# B&R Automation Studio project PloterCNC (part 5)

```c
	return fmi2OK;
}
/* END: fmi2SetString */
/*****************************************************************************/

/*****************************************************************************/
/* BEGIN: fmi2GetFMUstate */
/*****************************************************************************/
/* Storage structure:
		State id (hard coded value)
		Data length (bytes)
		ModelInstance
		Real data storage
		Integer data storage
		Real backup data storage (only for ME)
		Jacobian storage
		Error code
		String storage
*/
#define FMUStateID 983472598

fmi2Status fmi2GetFMUstate (
	fmi2Component	c,
	fmi2FMUstate*	FMUstate
)
{
	ModelInstance* comp = (ModelInstance *)c;
	char *cur;
	fmi2Real *rcur;
	M_INT i,j,*icur,wsto,ssto,jsto,totsto;

	if (invalidState(comp, "fmi2GetFMUstate", modelInitialized))
		return fmi2Error;

	if(comp->fmuType==fmi2ModelExchange)
		wsto = NUMBER_OF_REALS*sizeof(fmi2Real);
	else
		wsto = 0;

#ifdef FMI2_PROVIDES_DERIVATIVES
	jsto=( (1+NDIFF+NINP)*(NDIFF+NOUT) + NIUNK*(NIKNO+1) )*sizeof(fmi2Real);
#else
	jsto=0;
#endif

	ssto=0;
	for(i=0;i<NUMBER_OF_STRINGS;i++)
		if(comp->s[i])
			ssto+=strlen(comp->s[i])+1;
		else
			ssto++;

	totsto = 2*sizeof(M_INT) +
				sizeof(ModelInstance) +
				NUMBER_OF_REALS*sizeof(fmi2Real) +
				NUMBER_OF_INTEGERS*sizeof(M_INT) +
				wsto +
				jsto +
				sizeof(M_INT) +
				ssto;

	/* Verify that previously allocated FMU state is of sufficient size */
	if(*FMUstate) {
		icur=(M_INT *)(*FMUstate);
		if(icur[0]!=FMUStateID) {
			/* FMUstate pointer is not previously allocated in this routine
				so no way to verify the size */
			compLog(compEnv, comp->instanceName, fmi2Warning, "warning",
				"fmi2GetFMUstate: called with non-NULL state pointer of unknown size. Assuming sufficiently large.");
		}
		else if(icur[1]<totsto) {
			comp->functions.freeMemory(*FMUstate);
			*FMUstate=NULL;
		}
	}

	if(*FMUstate==NULL)
		FMUstate[0] = (fmi2FMUstate)comp->functions.allocateMemory(1,totsto);

	cur = (char *)(*FMUstate);

	icur = (M_INT *)cur;
	icur[0] = FMUStateID;
	icur[1] = totsto;
	cur += 2*sizeof(M_INT);

	memcpy(cur,comp,sizeof(ModelInstance));
	cur += sizeof(ModelInstance);

	rcur = (fmi2Real*)cur;
	for (i=0;i<NUMBER_OF_REALS;i++)	rcur[i] = comp->S.w[i];
	cur += NUMBER_OF_REALS*sizeof(fmi2Real);

	icur = (M_INT *)cur;
	for (i=0;i<NUMBER_OF_INTEGERS;i++) icur[i] = comp->S.iw[i];
	cur += NUMBER_OF_INTEGERS*sizeof(M_INT);

	if(comp->fmuType==fmi2ModelExchange) {
		rcur = (fmi2Real*)cur;
		for (i=0;i<NUMBER_OF_REALS;i++)	rcur[i] = comp->S.wset[i];
		cur += NUMBER_OF_REALS*sizeof(fmi2Real);
	}

#ifdef FMI2_PROVIDES_DERIVATIVES
	rcur = (fmi2Real*)cur;
	for (i=0;i<(1+NDIFF+NINP)*(NDIFF+NOUT);i++)	rcur[i] = comp->Jacobian[i];
	cur += (1+NDIFF+NINP)*(NDIFF+NOUT)*sizeof(fmi2Real);

	rcur = (fmi2Real*)cur;
	for (i=0;i<NIUNK*NIKNO;i++)	rcur[i] = comp->initJacobian[i];
	cur += NIUNK*NIKNO*sizeof(fmi2Real);

	rcur = (fmi2Real*)cur;
	for (i=0;i<NIUNK;i++)	rcur[i] = comp->initRes[i];
	cur += NIUNK*sizeof(fmi2Real);
#endif

	icur = (M_INT *)cur;
	icur[0] = errorOccured;
	cur += sizeof(M_INT);

	for(i=0;i<NUMBER_OF_STRINGS;i++) {
		if(comp->s[i]) {
			for(j=0;comp->s[i][j]!='\0';j++)
				*(cur++)=comp->s[i][j];
		}
		*(cur++)='\0';
	}

	return fmi2OK;
}
/* END: fmi2GetFMUstate */
/*****************************************************************************/

/*****************************************************************************/
/* BEGIN: fmi2SetFMUstate */
/*****************************************************************************/
fmi2Status fmi2SetFMUstate (fmi2Component	c,
							fmi2FMUstate	FMUstate) {
	ModelInstance* comp = (ModelInstance *)c;
	char *cur;
	fmi2String *scur;
	fmi2Real *rcur,*wcur,*jcur1,*jcur2,*jcur3;
	M_INT i,j,l,*icur;

	if (invalidState(comp, "fmi2SetFMUstate", modelInitialized))
		return fmi2Error;

	cur = (char *)FMUstate;
	icur = (M_INT *)cur;
	if(icur[0]!=FMUStateID) {
		compLog(compEnv, comp->instanceName, fmi2Error, "error",
			"fmi2SetFMUstate: called with invalid FMUstate");
		return(fmi2Error);
	}
	cur += 2*sizeof(M_INT);

	rcur = comp->S.w;
	icur = comp->S.iw;
	wcur = comp->S.wset;
	jcur1 = comp->Jacobian;
	jcur2 = comp->initJacobian;
	jcur3 = comp->initRes;
	scur = comp->s;
	memcpy(comp,cur,sizeof(ModelInstance));
	comp->S.w  = rcur;
	comp->S.iw = icur;
	comp->S.wset = wcur;
	comp->Jacobian = jcur1;
	comp->initJacobian = jcur2;
	comp->initRes = jcur3;
	comp->s = scur;
	cur += sizeof(ModelInstance);

	rcur = (fmi2Real *)cur;
	for(i=0;i<NUMBER_OF_REALS;i++) comp->S.w[i] = rcur[i];
	cur += NUMBER_OF_REALS*sizeof(fmi2Real);

	icur = (M_INT *)cur;
	for (i=0;i<NUMBER_OF_INTEGERS;i++) comp->S.iw[i] = icur[i];
	cur += NUMBER_OF_INTEGERS*sizeof(M_INT);

	if(comp->fmuType==fmi2ModelExchange) {
		rcur = (fmi2Real *)cur;
		for(i=0;i<NUMBER_OF_REALS;i++) comp->S.wset[i] = rcur[i];
		cur += NUMBER_OF_REALS*sizeof(fmi2Real);
	}
	else
		comp->S.wset = NULL;

#ifdef FMI2_PROVIDES_DERIVATIVES
	rcur = (fmi2Real*)cur;
	for (i=0;i<(1+NDIFF+NINP)*(NDIFF+NOUT);i++)	comp->Jacobian[i] = rcur[i];
	cur += (1+NDIFF+NINP)*(NDIFF+NOUT)*sizeof(fmi2Real);

	rcur = (fmi2Real*)cur;
	for (i=0;i<NIUNK*NIKNO;i++)	comp->initJacobian[i] = rcur[i];
	cur += NIUNK*NIKNO*sizeof(fmi2Real);

	rcur = (fmi2Real*)cur;
	for (i=0;i<NIUNK;i++)	comp->initRes[i] = rcur[i];
	cur += NIUNK*sizeof(fmi2Real);
#else
	comp->Jacobian = NULL;
	comp->initJacobian = NULL;
	comp->initRes = NULL;
#endif

	icur = (M_INT *)cur;
	errorOccured = icur[0];
	cur += sizeof(M_INT);

	for(i=0;i<NUMBER_OF_STRINGS;i++) {
		l=(comp->s[i]) ? strlen(comp->s[i]) : 0;
		j=strlen(cur);
		if(j>l) {
			if(comp->s[i]) comp->functions.freeMemory((char *)comp->s[i]);
			comp->s[i]=(fmi2String)comp->functions.allocateMemory(1,j+1);
		}
		strcpy((char *)comp->s[i],cur);
		cur += j+1;
	}

	return fmi2OK;
}
/* END: fmi2SetFMUstate */
/*****************************************************************************/

/*****************************************************************************/
/* BEGIN: fmi2FreeFMUstate */
/*****************************************************************************/
fmi2Status fmi2FreeFMUstate(fmi2Component c,
							fmi2FMUstate* FMUstate) {
	ModelInstance* comp = (ModelInstance *)c;
	M_INT *icur;

	if (invalidState(comp, "fmi2FreeFMUstate",
		modelInstantiated|modelInitialized|modelTerminated|modelError))
		return fmi2Error;

	if( *FMUstate ) {
		icur = (M_INT *)(*FMUstate);
		if(icur[0]!=FMUStateID)
			compLog(compEnv, comp->instanceName, fmi2Warning, "warning",
				"fmi2FreeFMUstate: called with invalid FMUstate");
		comp->functions.freeMemory(*FMUstate);
	}

	*FMUstate = NULL;

	return fmi2OK;
}
/* END: fmi2FreeFMUstate */
/*****************************************************************************/

/*****************************************************************************/
/* BEGIN: fmi2SerializedFMUstateSize */
/*****************************************************************************/
fmi2Status fmi2SerializedFMUstateSize(	fmi2Component	c,
										fmi2FMUstate	FMUstate,
										size_t			*size) {
	ModelInstance* comp = (ModelInstance *)c;
	M_INT *icur;

	if (invalidState(comp, "fmi2SerializedFMUstateSize", modelInitialized))
		return fmi2Error;

	icur = (M_INT *)FMUstate;
	if(icur[0]!=FMUStateID) {
		compLog(compEnv, comp->instanceName, fmi2Error, "error",
			"fmi2SerializedFMUstateSize: called with invalid FMUstate");
		return(fmi2Error);
	}
	*size = (size_t)icur[1];

	return fmi2OK;
}
/* END: fmi2SerializedFMUstateSize */
/*****************************************************************************/

/*****************************************************************************/
/* BEGIN: fmi2SerializeFMUstate */
/*****************************************************************************/
fmi2Status fmi2SerializeFMUstate(fmi2Component		c,
								fmi2FMUstate		FMUstate,
								fmi2Byte 			serializedState[],
								size_t				size) {
	ModelInstance* comp = (ModelInstance *)c;
	M_INT *icur;

	if (invalidState(comp, "fmi2SerializeFMUstate", modelInitialized))
		return fmi2Error;

	icur = (M_INT *)FMUstate;
	if(icur[0]!=FMUStateID) {
		compLog(compEnv, comp->instanceName, fmi2Error, "error",
			"fmi2SerializedFMUstate: called with invalid FMUstate");
		return fmi2Error;
	}
	if(icur[1]>(M_INT)size) {
		compLog(compEnv, comp->instanceName, fmi2Error, "error",
			"fmi2SerializedFMUstate: called with size not sufficient to contain FMUstate");
		return fmi2Error;
	}
	memcpy(serializedState, FMUstate, size);

	return fmi2OK;
}
/* END: fmi2SerializeFMUstate */
/*****************************************************************************/

/*****************************************************************************/
/* BEGIN: fmi2DeSerializeFMUstate */
/*****************************************************************************/
fmi2Status fmi2DeSerializeFMUstate(	fmi2Component	c,
									const fmi2Byte	serializedState[],
									size_t			size,
									fmi2FMUstate	*FMUstate) {
	ModelInstance* comp = (ModelInstance *)c;
	M_INT *icur;

	if (invalidState(comp, "fmi2DeSerializeFMUstate", modelInitialized))
		return fmi2Error;

	icur = (M_INT *)serializedState;
	if(icur[0]!=FMUStateID) {
		compLog(compEnv, comp->instanceName, fmi2Error, "error",
			"fmi2DeSerializedFMUstate: called with serializedState not containing valid FMUstate");
		return fmi2Error;
	}
	if(icur[1]>(M_INT)size) {
		compLog(compEnv, comp->instanceName, fmi2Error, "error",
			"fmi2SerializedFMUstate: called with size not sufficient to contain serializedState");
		return fmi2Error;
	}
	FMUstate[0] = (fmi2FMUstate)comp->functions.allocateMemory(1,size);
	memcpy(*FMUstate, serializedState, size);

	return fmi2OK;
}
/* END: fmi2DeSerializeFMUstate */
/*****************************************************************************/

/*****************************************************************************/
/* BEGIN: fmi2GetDirectionalDerivative */
/*****************************************************************************/
fmi2Status fmi2GetDirectionalDerivative(	fmi2Component			c,
										const fmi2ValueReference	vUnknown_ref[],
										size_t						nUnknown,
										const fmi2ValueReference	vKnown_ref[],
										size_t						nKnown,
										const fmi2Real				dvKnown[],
										fmi2Real					dvUnknown[]) {
#ifdef FMI2_PROVIDES_DERIVATIVES
	int i, j, k, row, col, offset;
	fmi2Status sts;
	fmi2ValueReference vrs, vrd;
	ModelInstance* comp = (ModelInstance *)c;

	if (invalidState(comp, "fmi2GetDirectionalDerivatives", modelInstantiated|modelInitialized))
		return fmi2Error;
	if (nKnown>0 && nullPointer(comp, "fmi2GetDirectionalDerivative", "vKnown_ref[]", vKnown_ref))
		return fmi2Error;
	if (nUnknown>0 && nullPointer(comp, "fmi2GetDirectionalDerivative", "vUnknown_ref[]", vUnknown_ref))
		return fmi2Error;
	if (nKnown>0 && nullPointer(comp, "fmi2GetDirectionalDerivative", "dvKnown[]", dvKnown))
		return fmi2Error;

	sts = syncModel(comp,"fmi2GetDirectionalDerivative");
	if ( sts!=fmi2OK ) return sts;

	/* Initialize unknown vector */
	for (i=0; i<nUnknown; i++) dvUnknown[i] = 0.;

	/* Get Jacobian information, dimensions, data, etc? */
	if(!comp->jsynced) {
		if(comp->initializeMode)
			initjac(comp->S.w[0],&(comp->S.w[1]),&(comp->S.w[NEQ+NPAR+1]),comp->initRes,comp->initJacobian);
		else
			intjac(comp->S.w[0],&(comp->S.w[1]),&(comp->S.w[NEQ+NPAR+1]),comp->Jacobian);
		comp->jsynced = fmi2True;
	}

	/* Order of value references :
	t, #states, #index-1(inps), #discrete, #params, #derivs, #events */

	/* Start the computation loop */
	if (comp->initializeMode) {
		offset = NIKNO;
		for (i=0; i<nKnown; i++) {
			/* Check the seed */
			if (dvKnown[i]!=0) {
				vrs = vKnown_ref[i];
				/* assert(vr>=0 && vr<NUMBER_OF_REALS); */
				col = -1;
				for (k=0; k<NIKNO; k++)
					if (vrs==vrIknowns[k]) {
						col = k;
						break;
					}
				/* Compute column i */
				for (j=0; j<nUnknown; j++) {
					vrd = vUnknown_ref[j];
					/* assert(vrd>=0 && vrd<NUMBER_OF_REALS); */
					if ( vrd==vrs ) {
						dvUnknown[j] += 1.0;
					}
					else if(col!=-1) {
						for (k=0; k<NIUNK; k++)
							if (vrd==vrIunknowns[k]) {
								dvUnknown[j] += dvKnown[i]*comp->initJacobian[k*offset+col];
								break;
							}
					}
				}
			}
		}
	}
	else {
		offset = 1+NDIFF+NINP;
		for (i=0; i<nKnown; i++) {
			/* Check the seed */
			if (dvKnown[i]!=0) {
				vrs = vKnown_ref[i];
				/* assert(vr>=0 && vr<NUMBER_OF_REALS); */
				/* Check that vKnown_ref[i] is a state or input */
				if ( vrs==0 || (vrs>=vrStates[0] && vrs<vrStates[0]+NDIFF) )
					col = vrs;
				else if(vrs>=1+NDIFF+NIX1-NINP && vrs<1+NDIFF+NIX1)
					col = vrs-(NIX1-NINP);
				else
					return fmi2Error;
				/* Compute column i */
				for (j=0; j<nUnknown; j++) {
					vrd = vUnknown_ref[j];
					/* assert(vrd>=0 && vrd<NUMBER_OF_REALS); */
					/* Check if vrd is a derivative or an output,
					it could also be an output that's a state */
					if ( vrd>=vrDers[0] && vrd<vrDers[0]+NDIFF ) {
						row = vrd-vrDers[0];
						dvUnknown[j] += dvKnown[i]*comp->Jacobian[row*offset+col];
					}
					else if( vrd>=vrStates[0] && vrd<vrStates[0]+NDIFF ) {
						if ( vrd==vrs ) dvUnknown[j] += 1.0;
					}
					else {
						for (k=0; k<NOUT; k++)
							if (vrd==vrOuts[k]) {
								/* refval-t-states+derivs: vrd-1-NDIFF+NDIFF */
								row = vrd-1;
								dvUnknown[j] += dvKnown[i]*comp->Jacobian[row*offset+col];
								break;
							}
						if (k==NOUT) return fmi2Error;
					}
				}
			}
		}
	}
	return fmi2OK;
#else
	/* Compiler warning fix */
	int i=nUnknown+nKnown;
	void *tmp;
	tmp=(void *)vUnknown_ref;
	tmp=(void *)vKnown_ref;
	tmp=(void *)dvKnown;
	tmp=(void *)dvUnknown;
	if(i>0) tmp=(void *)c;
	i=((int *)tmp)[0];
	/* End compiler warning fix */
	return fmi2Error;
#endif
}
/* END: fmi2GetDirectionalDerivative */
/*****************************************************************************/

#if NCON>0 && defined(WMI_PROJECTION)
/*****************************************************************************/
/* BEGIN: fmi2Projection */
/*****************************************************************************/
fmi2Status fmi2Projection(	fmi2Component	c,
								fmi2Real	P[],
								fmi2Real	projectionTolerance,
								size_t	iterationLimit,
								fmi2Boolean	apply) {
	int i;
	fmi2Status sts;
	fmi2Real S2[NDIFF];

	ModelInstance* comp = (ModelInstance *)c;

	if (invalidState(comp, "fmi2Projection", modelInstantiated|modelInitialized))
		return fmi2Error;

	sts = syncModel(comp,"fmi2Projection");
	if ( sts!=fmi2OK ) return sts;

	for(i=0;i<NDIFF;i++) S2[i] = comp->S.w[i+1];
	i=Projection(comp->S.w[0], &comp->S.w[1], projectionTolerance,
		iterationLimit, NULL, comp->S.psto);
	if( i!=0 ){
		/* Restore state */
		for(i=0;i<NDIFF;i++) comp->S.w[i+1]=S2[i];
		return fmi2Discard;
	}
	for(i=0;i<NDIFF;i++) P[i] = comp->S.w[i+1]-S2[i];

	if( !apply ){
		for(i=0;i<NDIFF;i++) comp->S.w[i+1]=S2[i];
	}

	return fmi2OK;
}
/* END: fmi2Projection */
/*****************************************************************************/

/*****************************************************************************/
/* BEGIN: fmi2ProjectionStep: No longer supported */
/*****************************************************************************/
fmi2Status fmi2ProjectionStep(  fmi2Component	c,
								fmi2Real	S[]) {
	UNUSED(c);
	UNUSED(S);
	return fmi2Error;
}
/* END: fmi2ProjectionStep */
/*****************************************************************************/

/*****************************************************************************/
/* BEGIN: fmi2Constraint */
/*****************************************************************************/
fmi2Status fmi2Constraint(	fmi2Component	c,
								fmi2Real	C[]) {
	int cb, cr, nblk;
	fmi2Real blkdata[2];
	fmi2Status sts;

	ModelInstance* comp = (ModelInstance *)c;

	if (invalidState(comp, "fmi2Constraint", modelInstantiated|modelInitialized))
		return fmi2Error;

	sts = syncModel(comp,"fmi2Constraint");
	if ( sts!=fmi2OK ) return sts;

	/* Iterate over Residual blocks */
	Rblkp(comp->S.w[0], &comp->S.w[1], blkdata, 0, 0);
	nblk = (int)(blkdata[0]);
	cr = 0;
	for(cb=1;cb<=nblk;cb++) {
		Rblkp(comp->S.w[0], &comp->S.w[1], &C[cr], cb, 3);
		Rblkp(comp->S.w[0], &comp->S.w[1], blkdata, cb, 1);
		cr += (int)(blkdata[0]);
	}

	return fmi2OK;
}
/* END: fmi2Constraint */
/*****************************************************************************/

/*****************************************************************************/
/* BEGIN: fmi2ConstraintJacobian: No longer supported */
/*****************************************************************************/
fmi2Status fmi2ConstraintJacobian(	fmi2Component	c,
										fmi2Real	J[]) {

	/* If this function is required at some point, the code will need to be
	modified to fill in the ncon x ndiff Matrix using a sequence of calls to
	the block-based Jacobian. It is known that this will provide 0 entries
	for block dependencies on vars from a prior block, but this will only
	slow convergence of a newton approach, and be irrelevant when sufficiently
	close to the solution manifold */
	UNUSED(c);
	UNUSED(J);
	return fmi2Error;
}
/* END: fmi2ConstraintJacobian */
/*****************************************************************************/
#endif

#ifdef FMI2_COSIMULATION
/*****************************************************************************
 * FMI functions: only for FMI Co-Simulation 2.0
 *****************************************************************************/
/*****************************************************************************/
/* BEGIN: fmi2SetRealInputDerivatives */
fmi2Status fmi2SetRealInputDerivatives(	fmi2Component			c,
										const fmi2ValueReference vr[],
										size_t					nvr,
										const fmi2Integer		order[],
										const fmi2Real			value[]) {
	ModelInstance* comp = (ModelInstance *)c;

	if (invalidState(comp, "fmi2SetRealInputDerivatives", modelInitialized))
		return fmi2Error;
	if (comp->loggingOn)
		compLog(compEnv, comp->instanceName, fmi2OK, "log",
				"fmi2SetRealInputDerivatives: nvr= %d", nvr);

	UNUSED(vr);
	UNUSED(order);
	UNUSED(value);
	compLog(NULL, comp->instanceName, fmi2Error, "warning",
			"fmi2SetRealInputDerivatives: ignoring function call."
			" This model cannot interpolate inputs: canInterpolateInputs = \"fmi2False\"");

	return fmi2Warning;
}
/* END: fmi2SetRealInputDerivatives */
/*****************************************************************************/

/*****************************************************************************/
/* BEGIN: fmi2GetRealOutputDerivatives */
fmi2Status fmi2GetRealOutputDerivatives(fmi2Component			c,
										const fmi2ValueReference vr[],
										size_t					nvr,
										const fmi2Integer		order[],
										fmi2Real				value[]) {
	int i;
	ModelInstance* comp = (ModelInstance *)c;

	if (invalidState(comp, "fmi2GetRealOutputDerivatives", modelInitialized))
		return fmi2Error;
	if (comp->loggingOn)
		compLog(compEnv, comp->instanceName, fmi2OK, "log",
				"fmi2GetRealOutputDerivatives: nvr= %d",	nvr);

	UNUSED(vr);
	UNUSED(order);
	compLog(NULL, comp->instanceName, fmi2Error, "warning",
			"fmi2GetRealOutputDerivatives: ignoring function call."
			" This model cannot compute derivatives of outputs: MaxOutputDerivativeOrder=\"0\"");

	for (i=0; i<(int)nvr; i++) value[i] = 0;

	return fmi2Warning;
}
/* END: fmi2GetRealOutputDerivatives */
/*****************************************************************************/

#define MAX_STEP  1.00000000000000000e-04

/*****************************************************************************/
/* BEGIN: fmi2DoStep */
fmi2Status fmi2DoStep(  fmi2Component	c,
						fmi2Real		currentCommunicationPoint,
						fmi2Real		communicationStepSize,
						fmi2Boolean		newStep) {

	ModelInstance* comp	= (ModelInstance *)c;
	int		i;
	double	h;
#if NEVT>0
	M_INT *modes;
	double	prevEventIndicators[max(NEVT, 1)];
#endif

	if (invalidState(comp, "fmi2DoStep", modelInitialized)) return fmi2Error;

	if (comp->loggingOn)
		compLog(compEnv, comp->instanceName, fmi2OK, "log", "fmi2DoStep: "
				"currentCommunicationPoint = %g, "
				"communicationStepSize = %g, "
				"newStep = fmi2%s",
				currentCommunicationPoint, communicationStepSize, newStep ? "True" : "False");

	if (comp->stopTimeDefined && currentCommunicationPoint+communicationStepSize > comp->stopTime) {
		comp->state = modelError;
		return fmi2Error;
	}

#if NPAR>0
	if(pchange) {
		SolverInitialize(&(comp->S));
		pchange=0;
		if (errorOccured>0) {
			setVidError(comp,NULL);
			if (comp->fptr) {
				writeErrorToFile(comp->fptr,NULL);
				comp->fptr = NULL;
			}
			comp->state = modelTerminated;
			logMessage(comp, "fmi2DoStep", "error", fmi2Error);
			return fmi2Error;
		}
		else if(errorOccured<0) {
			logMessage(comp, "fmi2DoStep", "warning", fmi2Warning);
			errorOccured=0;
		}
	}
#endif

#if NEVT>0
	/* Run to get initial event indicators */
	eev(comp->S.w[0],&(comp->S.w[1]),&(comp->S.w[1]),prevEventIndicators);
	modes=comp->S.iw;
	ComputeEventIndicators(prevEventIndicators,&(comp->S.w[1]),modes,
		&modes[3*NEVT],&modes[2*NEVT],&modes[4*NEVT]);
#endif

	comp->S.w[0] = currentCommunicationPoint;
	if( currentCommunicationPoint < (comp->lastSuccessfulTime-10.*ULP1) )
		comp->lastStepSize = -1.;
	h = ( comp->lastStepSize<0. ) ? communicationStepSize/100. : comp->lastStepSize;
	warningOccured=0;
	/* Call the variable step integrator */
	i = Integrate(comp->S.w,comp->S.iw,currentCommunicationPoint+communicationStepSize,
				ERRTOL,&h,comp->S.psto);
	if(warningOccured) {
		logWarning(comp, "Integrate", "warning", fmi2Warning);
		warningOccured=0;
	}
	if(i!=1) {
		if (errorOccured>0) {
			comp->state = modelTerminated;
			logMessage(comp, "fmi2DoStep", "error", fmi2Error);
			return fmi2Error;
		}
	}
	comp->lastStepSize = (fmi2Real)h;
	comp->synced = fmi2True;
	comp->jsynced = fmi2False;
	SolverOutputs(&(comp->S));

	comp->lastSuccessfulTime = currentCommunicationPoint + communicationStepSize;
	comp->vidsts = 2;
 	if (comp->fptr)
		fwrite(comp->S.w,sizeof(fmi2Real),NEQ+1,comp->fptr);

	return fmi2OK;
}
/* END: fmi2DoStep */
/*****************************************************************************/

/*****************************************************************************/
/* BEGIN: fmi2CancelStep */
fmi2Status fmi2CancelStep(fmi2Component c) {
	ModelInstance* comp = (ModelInstance *)c;

	if (invalidState(comp, "fmi2CancelStep", modelInitialized)) return fmi2Error;
	if (comp->loggingOn)
		compLog(compEnv, comp->instanceName, fmi2OK, "log", "fmi2CancelStep");

	compLog(NULL, comp->instanceName, fmi2Error, "error",
			"fmi2CancelStep: Can be called when fmi2DoStep returned fmi2Pending."
			" This is not the case.");
	comp->state = modelError;
	return fmi2Error;
}
/* END: fmi2CancelStep */
/*****************************************************************************/

/*****************************************************************************/
/* BEGIN: fmi2GetStatus */
fmi2Status fmi2GetStatus(	fmi2Component		c,
							const fmi2StatusKind s,
							fmi2Status*			value) {
	ModelInstance* comp = (ModelInstance *)c;

	if (invalidState(comp, "fmi2GetStatus", modelInstantiated|modelInitialized))
		return fmi2Error;

	UNUSED(value);
	if (s==fmi2DoStepStatus) {
		if (comp->loggingOn) {
			compLog(compEnv, comp->instanceName, fmi2OK, "log",
				"[fmi2GetStatus]: fmi2StatusKind = fmi2DoStepStatus");
			compLog(NULL, comp->instanceName, fmi2Error, "error",
				"[fmi2GetStatus]: Can be called with fmi2DoStepStatus when fmi2DoStep returned fmi2Pending."
				" This is not the case.");
		}
		return fmi2Discard;
	}
	else
		return fmi2Discard;
}
/* END: fmi2GetStatus */
/*****************************************************************************/

/*****************************************************************************/
/* BEGIN: fmi2GetRealStatus */
fmi2Status fmi2GetRealStatus(	fmi2Component		c,
								const fmi2StatusKind s,
								fmi2Real*			value) {
	ModelInstance* comp = (ModelInstance *)c;

	if (invalidState(comp, "fmi2GetRealStatus", modelInstantiated|modelInitialized))
		return fmi2Discard;

	if (s==fmi2LastSuccessfulTime) {
		if (comp->loggingOn) {
			compLog(compEnv, comp->instanceName, fmi2OK, "log",
				"[fmi2GetRealStatus]: fmi2StatusKind = fmi2LastSuccessfulTime");
		}
		if (comp->state==modelTerminated) {
			*value = comp->lastSuccessfulTime;
			return fmi2OK;
		}
		else {
			compLog(NULL, comp->instanceName, fmi2Error, "error",
				"[fmi2GetRealStatus]: Can be called with fmi2LastSuccessfulTime when fmi2DoStep returned fmi2Discard."
				" This is not the case.");
			return fmi2Discard;
		}
	}
	else
		return fmi2Discard;
}
/* END: fmi2GetRealStatus */
/*****************************************************************************/

/*****************************************************************************/
/* BEGIN: fmi2GetIntegerStatus */
fmi2Status fmi2GetIntegerStatus(fmi2Component		c,
								const fmi2StatusKind s,
								fmi2Integer*		value) {
	UNUSED(c);
	UNUSED(s);
	UNUSED(value);
	return fmi2Discard;
}
/* END: fmi2GetIntegerStatus */
/*****************************************************************************/

/*****************************************************************************/
/* BEGIN: fmi2GetBooleanStatus */
fmi2Status fmi2GetBooleanStatus(fmi2Component		c,
								const fmi2StatusKind s,
								fmi2Boolean*		value) {
	ModelInstance* comp = (ModelInstance *)c;

	if (invalidState(comp, "fmi2GetBooleanStatus", modelInstantiated|modelInitialized))
		return fmi2Discard;

	if (s==fmi2Terminated) {
		if (comp->loggingOn) {
			compLog(compEnv, comp->instanceName, fmi2OK, "log",
				"[fmi2GetBooleanStatus]: fmi2StatusKind = fmi2Terminated");
		}
		if (comp->state==modelTerminated)
			*value = fmi2True;
		else
			*value = fmi2False;
		return fmi2OK;
	}
	else
		return fmi2Discard;
}
/* END: fmi2GetBooleanStatus */
/*****************************************************************************/

/*****************************************************************************/
/* BEGIN: fmi2GetStringStatus */
fmi2Status fmi2GetStringStatus(	fmi2Component		c,
								const fmi2StatusKind s,
								fmi2String*			value) {
	ModelInstance* comp = (ModelInstance *)c;

	if (invalidState(comp, "fmi2GetStringStatus", modelInstantiated|modelInitialized))
		return fmi2Discard;

	UNUSED(value);
	if (s==fmi2PendingStatus) {
		if (comp->loggingOn) {
			compLog(compEnv, comp->instanceName, fmi2OK, "log",
				"[fmi2GetStringStatus]: fmi2StatusKind = fmi2PendingStatus");
			compLog(NULL, comp->instanceName, fmi2Error, "error",
					"[fmi2GetStringStatus]: Can be called with fmi2PendingStatus when fmi2DoStep returned fmi2Pending."
					" This is not the case.");
		}
		return fmi2Discard;
	}
	else
		return fmi2Discard;
}
/* END: fmi2GetStringStatus */
/*****************************************************************************/

#else
/*****************************************************************************
 * FMI functions: only for Model Exchange 2.0
 *****************************************************************************/

/*****************************************************************************/
/* BEGIN: fmi2EnterEventMode */
fmi2Status fmi2EnterEventMode(fmi2Component c) {
	ModelInstance* comp = (ModelInstance *)c;

	if (comp) {
		comp->lastEventTime = comp->S.w[0]-1.0;
		return fmi2OK;
	}
	else
		return fmi2Error;
}
/* END: fmi2EnterEventMode */
/*****************************************************************************/

/*****************************************************************************/
/* BEGIN: fmi2NewDiscreteStates */
fmi2Status fmi2NewDiscreteStates(fmi2Component	c,
								fmi2EventInfo*	eventInfo) {
	ModelInstance* comp = (ModelInstance *)c;
	int i;
#if NEVT+NCON>0
	fmi2Real save[NEQ],val;
#endif
	if (invalidState(comp, "fmi2NewDiscreteStates", modelInitialized))
		return fmi2Error;
	if (nullPointer (comp, "fmi2NewDiscreteStates", "eventInfo", eventInfo))
		return fmi2Error;

	eventInfo->newDiscreteStatesNeeded				= fmi2False;
	eventInfo->nominalsOfContinuousStatesChanged	= fmi2False;
	eventInfo->valuesOfContinuousStatesChanged		= fmi2False;
	eventInfo->terminateSimulation					= fmi2False;
	eventInfo->nextEventTimeDefined					= fmi2False;
	eventInfo->nextEventTime						= -0.0;

#if NEVT+NCON>0
	for(i=0;i<NEQ;i++) save[i]=comp->S.w[i+1];
#endif
	i=SolverProject(&(comp->S));
	if (i<0 || errorOccured==1) {
		setVidError(comp,NULL);
		if (comp->fptr) {
			writeErrorToFile(comp->fptr,NULL);
			comp->fptr = NULL;
		}
		eventInfo->terminateSimulation = fmi2True;
		comp->state = modelTerminated;
		logMessage(comp, "fmi2NewDiscreteStates", "error", fmi2Error);
		return fmi2Error;
	}
	else if (i>0 || errorOccured==2) {
		compLog(compEnv, comp->instanceName, fmi2OK, "log",
				"fmi2NewDiscreteStates: model requested termination at t = %g",
				comp->S.w[0]);
		setVidError(comp,NULL);
		if (comp->fptr) {
			writeErrorToFile(comp->fptr,NULL);
			comp->fptr = NULL;
		}
		eventInfo->terminateSimulation = fmi2True;
		comp->state = modelTerminated;
		logMessage(comp, "fmi2NewDiscreteStates", "warning", fmi2Discard);
		return fmi2OK;
	}
	else if(errorOccured<0) {
		logMessage(comp, "fmi2NewDiscreteStates", "warning", fmi2Warning);
		errorOccured=0;
	}
#if NEVT>0
	if (comp->S.w[0]!=comp->lastEventTime) {
		i=RunEvents(comp->S.w, comp->S.iw, 0, -1, EVTITER, comp->S.psto);
		if (i<0 || errorOccured==1) {
			setVidError(comp,NULL);
			if (comp->fptr) {
				writeErrorToFile(comp->fptr,NULL);
				comp->fptr = NULL;
			}
			eventInfo->terminateSimulation = fmi2True;
			comp->state = modelTerminated;
			logMessage(comp, "fmi2NewDiscreteStates", "error", fmi2Error);
			return fmi2Error;
		}
		else if (i>0 || errorOccured==2) {
			compLog(compEnv, comp->instanceName, fmi2OK, "log",
					"fmi2NewDiscreteStates: model requested termination at t = %g",
					comp->S.w[0]);
			setVidError(comp,NULL);
			if (comp->fptr) {
				writeErrorToFile(comp->fptr,NULL);
				comp->fptr = NULL;
			}
			eventInfo->terminateSimulation = fmi2True;
			comp->state = modelTerminated;
			logMessage(comp, "fmi2NewDiscreteStates", "warning", fmi2Discard);
			return fmi2OK;
		}
		else if(errorOccured<0) {
			logMessage(comp, "fmi2NewDiscreteStates", "warning", fmi2Warning);
			errorOccured=0;
		}
		comp->lastEventTime = comp->S.w[0];
	}
	i=RunEvents(comp->S.w, comp->S.iw, 1, -1, EVTITER, comp->S.psto);
	if (i<0 || errorOccured==1) {
		setVidError(comp,NULL);
		if (comp->fptr) {
			writeErrorToFile(comp->fptr,NULL);
			comp->fptr = NULL;
		}
		eventInfo->terminateSimulation = fmi2True;
		comp->state = modelTerminated;
		logMessage(comp, "fmi2NewDiscreteStates", "error", fmi2Error);
		return fmi2Error;
	}
	else if (i>0 || errorOccured==2) {
		compLog(compEnv, comp->instanceName, fmi2OK, "log",
				"fmi2NewDiscreteStates: model requested termination at t = %g",
				comp->S.w[0]);
		setVidError(comp,NULL);
		if (comp->fptr) {
			writeErrorToFile(comp->fptr,NULL);
			comp->fptr = NULL;
		}
		eventInfo->terminateSimulation = fmi2True;
		comp->state = modelTerminated;
		logMessage(comp, "fmi2NewDiscreteStates", "warning", fmi2Discard);
		return fmi2OK;
	}
	else if(errorOccured<0) {
		logMessage(comp, "fmi2NewDiscreteStates", "warning", fmi2Warning);
		errorOccured=0;
	}
#endif
#if NEVT+NCON>0
	for(i=0;i<NEQ;i++) {
		val=1e-15;
		if(fabs(save[i])>val) val=fabs(save[i]);
		if(fabs(comp->S.w[i+1])>val) val=fabs(comp->S.w[i+1]);
		if( fabs(comp->S.w[i+1]-save[i])>1e-12*val )
			eventInfo->valuesOfContinuousStatesChanged = fmi2True;
	}
	if(eventInfo->valuesOfContinuousStatesChanged==fmi2True)
		SolverOutputs(&(comp->S));
#endif
	return fmi2OK;
}
/* END: fmi2NewDiscreteStates */
/*****************************************************************************/

/*****************************************************************************/
/* BEGIN: fmi2EnterContinuousTimeMode */
fmi2Status fmi2EnterContinuousTimeMode(fmi2Component c) {
	if (c)	return fmi2OK;
	else	return fmi2Error;
}
/* END: fmi2EnterContinuousTimeMode */
/*****************************************************************************/

/*****************************************************************************/
/* BEGIN: fmi2CompletedIntegratorStep */
fmi2Status fmi2CompletedIntegratorStep(	fmi2Component	c,
										fmi2Boolean		noSetFMUStatePriorToCurrentPoint,
										fmi2Boolean*	enterEventMode,
										fmi2Boolean*	terminateSimulation) {
	ModelInstance* comp = (ModelInstance *)c;
	int i;
#if NCON>0 && defined(CONDSTEPEVENT)
	fmi2Real save[NEQ],val,drift;
#endif

	UNUSED(noSetFMUStatePriorToCurrentPoint);
	if (invalidState(comp, "fmi2CompletedIntegratorStep", modelInitialized))
		return fmi2Error;
	if (nullPointer (comp, "fmi2CompletedIntegratorStep", "enterEventMode", enterEventMode))
		return fmi2Error;
	if (nullPointer (comp, "fmi2CompletedIntegratorStep", "terminateSimulation", terminateSimulation))
		return fmi2Error;
	if (comp->loggingOn)
		compLog(compEnv, comp->instanceName, fmi2OK, "log",
				"fmi2CompletedIntegratorStep");

	*terminateSimulation = fmi2False;

	if (comp->synced)
		SolverUpdate(&(comp->S),1,1);
	else {
		SolverUpdate(&(comp->S),0,1);
		if (errorOccured>0) {
			setVidError(comp,NULL);
			if (comp->fptr) {
				writeErrorToFile(comp->fptr,NULL);
				comp->fptr = NULL;
			}
			errorOccured = 0;
			comp->state = modelTerminated;
			logMessage(comp, "fmi2CompletedIntegratorStep", "error", fmi2Discard);
			return fmi2Discard;
		}
		else if(errorOccured<0) {
			logMessage(comp, "fmi2CompletedIntegratorStep", "warning", fmi2Warning);
			errorOccured=0;
		}
		comp->synced = fmi2True;
		comp->jsynced = fmi2False;
	}
	if(comp->fmuType==fmi2ModelExchange && comp->S.wset)
		for(i=NDIFF+1;i<=NDIFF+NIX1-NINP;i++)
			comp->S.wset[i]=comp->S.w[i];
	SolverOutputs(&(comp->S));
	if( comp->S.w[0]>=(comp->vidlasttime+comp->minSampleStep)*(1-1e-15) ) {
		comp->vidsts=2;
		comp->vidlasttime=comp->S.w[0];
	}
 	if (comp->fptr)
		if ( comp->S.w[0]>=(comp->lastsampletime+comp->minSampleStep)*(1-1e-15) ) {
			fwrite(comp->S.w,sizeof(fmi2Real),NEQ+1,comp->fptr);
			comp->lastsampletime=comp->S.w[0];
			if ( comp->numpts++ == WARNNUMDATPTS )
				compLog(compEnv, comp->instanceName, fmi2Warning, "warning",
						"[fmi2CompletedIntegratorStep]: At time t=%.16g, %d data points were written into file %s; consider increasing the minimum sample step, %.16g, to limit file size.",
						comp->S.w[0], WARNNUMDATPTS, comp->fstr, comp->minSampleStep);
		}

#if !defined(WMI_PROJECTION) && NCON>0
#   if defined(CONDSTEPEVENT)
	for(i=0;i<NEQ;i++) save[i]=comp->S.w[i+1];
	i=SolverProject(&(comp->S));
	if (i<0 || errorOccured>=1) {
		errorOccured=0;
		*enterEventMode = fmi2True;
	}
	else if (i>0) {
		setVidError(comp,NULL);
		if (comp->fptr) {
			writeErrorToFile(comp->fptr,NULL);
			comp->fptr = NULL;
		}
		comp->state = modelTerminated;
		*terminateSimulation = fmi2True;
		logMessage(comp, "fmi2CompletedIntegratorStep", "error", fmi2Discard);
		return fmi2OK;
	}
	else {
		drift=0.0;
		for(i=0;i<NEQ;i++) {
			val=1e-15;
			if(fabs(save[i])>val) val=fabs(save[i]);
			if(fabs(comp->S.w[i+1])>val) val=fabs(comp->S.w[i+1]);
			val=fabs(comp->S.w[i+1]-save[i])/val;
			if(val>drift) drift=val;
		}
		val=(CONTOL<1e-8) ? 1e-10 : 0.01*CONTOL;
		if(drift>val)
			*enterEventMode = fmi2True;
		else
			*enterEventMode = fmi2False;
	}
	for(i=0;i<NEQ;i++) comp->S.w[i+1]=save[i];
#   else
	*enterEventMode = fmi2True;
#   endif
#else
	*enterEventMode = fmi2False;
#endif

	return fmi2OK;
}
/* END: fmi2CompletedIntegratorStep */
/*****************************************************************************/

/*****************************************************************************/
/* BEGIN: fmi2SetTime */
fmi2Status fmi2SetTime(	fmi2Component	c,
						fmi2Real		time) {
	ModelInstance* comp = (ModelInstance *)c;
	if (invalidState(comp, "fmi2SetTime", modelInstantiated|modelInitialized))
		return fmi2Error;
	if (comp->loggingOn)
		compLog(compEnv, comp->instanceName, fmi2OK, "log",
				"fmi2SetTime: time = %.16g", time);
	if (comp->S.w[0] != time) {
		comp->S.w[0] = time;
		comp->synced = fmi2False;
		comp->jsynced = fmi2False;
	}
	return fmi2OK;
}
/* END: fmi2SetTime */
/*****************************************************************************/

/*****************************************************************************/
/* BEGIN: fmi2SetContinuousStates */
fmi2Status fmi2SetContinuousStates(	fmi2Component	c,
									const fmi2Real	x[],
									size_t			nx){
	ModelInstance* comp = (ModelInstance *)c;
#if NDIFF>0
	double scalev;
	int i;
	fmi2ValueReference vr;
#endif

	if (invalidState (comp, "fmi2SetContinuousStates", modelInitialized))
		return fmi2Error;
	if (invalidNumber(comp, "fmi2SetContinuousStates", "nx", nx, NDIFF))
		return fmi2Error;
#if NDIFF>0
	if (nullPointer  (comp, "fmi2SetContinuousStates", "x[]", x))
		return fmi2Error;

	for (i=0; i<(int)nx; i++) {
		vr = vrStates[i];
		if (comp->loggingOn)
			compLog(compEnv, comp->instanceName, fmi2OK, "log",
					"fmi2SetContinuousStates: #r%d# = %.16g", vr, x[i]);
		/*assert(vr>=0 && vr<NUMBER_OF_REALS);*/
		if( nomfac )
			scalev = nomfac[i]*x[i];
		else
			scalev = x[i];
		if (comp->S.w[vr] != scalev) {
			comp->S.w[vr] = scalev;
			comp->synced = fmi2False;
			comp->jsynced = fmi2False;
		}
	}
#endif
	return fmi2OK;
}
/* END: fmi2SetContinuousStates */
/*****************************************************************************/

/*****************************************************************************/
/* BEGIN: fmi2GetDerivatives */
fmi2Status fmi2GetDerivatives(	fmi2Component	c,
								fmi2Real		derivatives[],
								size_t			nx) {
#if NDIFF>0
	int i;
#endif
	ModelInstance* comp = (ModelInstance *)c;

	if (invalidState (comp, "fmi2GetDerivatives", validGet))
		return fmi2Error;
	if (invalidNumber(comp, "fmi2GetDerivatives", "nx", nx, NDIFF))
		return fmi2Error;
	if (nullPointer  (comp, "fmi2GetDerivatives", "derivatives[]", derivatives))
		return fmi2Error;

#if NDIFF>0
	if (comp->state==modelInitialized && !comp->synced) {
		SolverUpdate(&(comp->S),0,0);
		if(errorOccured>0) {
			setVidError(comp,NULL);
			if (comp->fptr) {
				writeErrorToFile(comp->fptr,NULL);
				comp->fptr = NULL;
			}
			errorOccured=0;
			logMessage(comp, "fmi2GetDerivatives", "error", fmi2Discard);
			return fmi2Discard;
		}
		else if(errorOccured<0) {
			logMessage(comp, "fmi2GetDerivatives", "warning", fmi2Warning);
			errorOccured=0;
		}
		comp->synced = fmi2True;
		comp->jsynced = fmi2False;
	}
	for (i=0; i<(int)nx; i++) {
		if( nomfac )
			derivatives[i] = comp->S.w[vrDers[i]]/nomfac[i];
		else
			derivatives[i] = comp->S.w[vrDers[i]];
		if (comp->loggingOn)
			compLog(compEnv, comp->instanceName, fmi2OK, "log",
					"fmi2GetDerivatives: #r%d# = %.16g",	vrDers[i], derivatives[i]);
	}
#endif
	return fmi2OK;
}
/* END: fmi2GetDerivatives */
/*****************************************************************************/

/*****************************************************************************/
/* BEGIN: fmi2GetEventIndicators */
fmi2Status fmi2GetEventIndicators(	fmi2Component	c,
									fmi2Real		eventIndicators[],
									size_t			ni) {
#if NEVT>0
	int i;
	M_INT *modes;
	fmi2Status sts;
#endif
	ModelInstance* comp = (ModelInstance *)c;

	if (invalidState (comp, "fmi2GetEventIndicators", validGet))
		return fmi2Error;
	if (invalidNumber(comp, "fmi2GetEventIndicators", "ni", ni, NEVT))
		return fmi2Error;

#if NEVT>0
	sts = syncModel(c,"fmi2GetEventIndicators");
	if ( sts!=fmi2OK ) return(sts);
	eev(comp->S.w[0],&(comp->S.w[1]),&(comp->S.w[1]),eventIndicators);
	modes=comp->S.iw;
	ComputeEventIndicators(eventIndicators,&(comp->S.w[1]),modes,
		&modes[3*NEVT],&modes[2*NEVT],&modes[4*NEVT]);
	for (i=0; i<(int)ni; i++) {
		if (comp->loggingOn)
			compLog(compEnv, comp->instanceName, fmi2OK, "log",
					"fmi2GetEventIndicators: z%d = %.16g",
					i, eventIndicators[i]);
	}
#else
	UNUSED(eventIndicators);
#endif
	return fmi2OK;
}
/* END: fmi2GetEventIndicators */
/*****************************************************************************/

/*****************************************************************************/
/* BEGIN: fmi2GetContinuousStates */
fmi2Status fmi2GetContinuousStates(	fmi2Component	c,
									fmi2Real		states[],
									size_t			nx) {
#if NDIFF>0
	int i;
	fmi2Status sts;
#endif
	ModelInstance* comp = (ModelInstance *)c;

	if (invalidState (comp, "fmi2GetContinuousStates", validGet))
		return fmi2Error;
	if (invalidNumber(comp, "fmi2GetContinuousStates", "nx", nx, NDIFF))
		return fmi2Error;
#if NDIFF>0
	if (nullPointer  (comp, "fmi2GetContinuousStates", "states[]", states))
		return fmi2Error;

	sts = syncModel(c,"fmi2GetContinuousStates");
	if ( sts!=fmi2OK ) return(sts);
	for (i=0; i<(int)nx; i++) {
		if( nomfac )
			states[i] = comp->S.w[vrStates[i]]/nomfac[i];
		else
			states[i] = comp->S.w[vrStates[i]];
		if (comp->loggingOn)
			compLog(compEnv, comp->instanceName, fmi2OK, "log",
					"fmi2GetContinuousStates: #r%u# = %.16g", vrStates[i], states[i]);
	}
#endif
	return fmi2OK;
}
/* END: fmi2GetContinuousStates */
/*****************************************************************************/

/*****************************************************************************/
/* BEGIN: fmi2GetNominalsOfContinuousStates */
fmi2Status fmi2GetNominalsOfContinuousStates(fmi2Component	c,
											fmi2Real		x_nominal[],
											size_t			nx) {
	ModelInstance* comp = (ModelInstance *)c;
	int i;

	if (invalidState (comp, "fmi2GetNominalsOfContinuousStates", validGet))
		return fmi2Error;
	if (invalidNumber(comp, "fmi2GetNominalsOfContinuousStates", "nx", nx, NDIFF))
		return fmi2Error;
	if (nullPointer  (comp, "fmi2GetNominalsOfContinuousStates", "x_nominal[]", x_nominal))
		return fmi2Error;

	if (comp->loggingOn)
		compLog(compEnv, comp->instanceName, fmi2OK, "log",
				"fmi2GetNominalsOfContinuousStates: x_nominal[0..%d] = 1.0", nx-1);
	if( nomfac )
		for (i=0; i<(int)nx; i++) x_nominal[i] = 1.0/nomfac[i-1];
	else
		for (i=0; i<(int)nx; i++) x_nominal[i] = 1.0;

	return fmi2OK;
}
/* END: fmi2GetNominalsOfContinuousStates */
/*****************************************************************************/

#endif

/*****************************************************************************/
/* Special purpose data communication functions */

typedef fmi2Status getMapleSimVideoDataLengthTYPE(fmi2Component, fmi2Integer *);
#define getMapleSimVideoDataLength fmi2FullName(getMapleSimVideoDataLength)
FMI2_Export getMapleSimVideoDataLengthTYPE getMapleSimVideoDataLength;

fmi2Status getMapleSimVideoDataLength(fmi2Component c, fmi2Integer *len)
{
	ModelInstance* comp = (ModelInstance *)c;

	if(comp->vidsts==0) {
		*len=0;
		return(fmi2Warning);
	}
	else if(comp->vidsts==1)
		*len=2+NPAR;
	else if(comp->vidsts==2)
		*len=NEQ+1;
	else if(comp->vidsts==-1)
		*len=2+strlen(comp->viderror)/8;
	else {
		*len=0;
		return(fmi2Error);
	}
	return(fmi2OK);
}

typedef fmi2Status getMapleSimVideoDataTYPE(fmi2Component, fmi2Real *);
#define getMapleSimVideoData fmi2FullName(getMapleSimVideoData)
FMI2_Export getMapleSimVideoDataTYPE getMapleSimVideoData;

fmi2Status getMapleSimVideoData(fmi2Component c, fmi2Real *data)
{
	ModelInstance* comp = (ModelInstance *)c;

	if(comp->vidsts==0)
		return(fmi2Error);
	else if(comp->vidsts==1) {
		data[0]=nData[0];
		data[1]=nData[1];
		memcpy(&data[2],&comp->S.w[NEQ+1],NPAR*sizeof(fmi2Real));
	}
	else if(comp->vidsts==2)
		memcpy(data,comp->S.w,(NEQ+1)*sizeof(fmi2Real));
	else if(comp->vidsts==-1) {
		data[0]=-1e10;
		memcpy(&data[1],comp->viderror,strlen(comp->viderror)+1);
	}
	else
		return(fmi2Error);
	comp->vidsts=0;
	return(fmi2OK);
}

typedef fmi2Status getMapleSimAuxiliaryDataTYPE(fmi2Component, fmi2Real *);
#define getMapleSimAuxiliaryData fmi2FullName(getMapleSimAuxiliaryData)
FMI2_Export getMapleSimAuxiliaryDataTYPE getMapleSimAuxiliaryData;

fmi2Status getMapleSimAuxiliaryData(fmi2Component c, fmi2Real *data)
{
	ModelInstance* comp = (ModelInstance *)c;

	if(!comp->synced) {
		auxp(comp->S.w[0],&(comp->S.w[1]),&(comp->S.w[NEQ+NPAR+1]),data);
		return(fmi2Discard);
	}
	else if(comp->state==modelInitialized) {
		auxp(comp->S.w[0],&(comp->S.w[1]),&(comp->S.w[NEQ+NPAR+1]),data);
		return(fmi2OK);
	}
	else return(fmi2Error);
}
```

#### CNC_FMUFmiSceneView.c
```c
#include <bur/plctypes.h>
#include <sys_lib.h>
#include "CNC_FMULib.h"

#include <fmi2Functions.h>

#include <stdlib.h>
#include <stdio.h>
#include <string.h>
#include <math.h>

void CNC_FMUView(struct CNC_FMUView* fubInstance)
{
	if (fubInstance->Enable == 1) {

		if (fubInstance->InstRef->Fmi2.Enabled) {
			CNC_FMU_getMapleSimAuxiliaryData(fubInstance->InstRef->Fmi2.Instance, &(fubInstance->vInternal));
		}

		int i;
		for (i=0; i <= 18; i++) {
			fubInstance->ObjPos[i] = (float)fubInstance->vInternal[i];
		}

		} else {

	}

}
```

#### CNC_FMUImpl.c
```c
/********************************************************************
 * COPYRIGHT -- Bernecker + Rainer
 ********************************************************************

 ********************************************************************
 * Basic fmu/fub implementation
 ********************************************************************/

#include <bur/plctypes.h>
#include <sys_lib.h>
#include <fmi2Functions.h>

#ifdef __cplusplus
	extern "C"
	{
#endif
#include "CNC_FMULib.h"
#ifdef __cplusplus
	};
#endif

/**********************************************************************/
/* FUB interface declarations */
#define  FMU_Enable 			fubInstance->Enable

#define  FMU_Instance 			fubInstance->Internal.Fmi2.Instance
#define  FMU_Enabled 			fubInstance->Internal.Fmi2.Enabled
#define  FMU_Error 			fubInstance->Internal.Fmi2.Error
#define  FMU_EndTime    		fubInstance->Internal.Fmi2.EndTime
#define  FMU_StartTime    		fubInstance->Internal.Fmi2.StartTime
#define  FMU_CurrentTime   		fubInstance->Internal.Fmi2.CurrentTime
#define  FMU_StepSize    		fubInstance->Internal.Fmi2.StepSize
#define  FMU_Callbacks   		fubInstance->Internal.Fmi2.Callbacks

/**********************************************************************/
/* Method delcarations */
void CNC_FMU_fmuLogger(fmi2Component c, fmi2String instanceName, fmi2Status status, fmi2String category, fmi2String message, ...);
void* CNC_FMU_AllocateMemory(UDINT numElements, UDINT elementSize);
void CNC_FMU_FreeMemory(void* pMemory);

void CNC_FMU_initFMU(struct CNC_FMU* fubInstance);

void CNC_FMU_initFMUCallbacks(struct CNC_FMU* fubInstance);
void CNC_FMU_initFMUCoSimParameters(struct CNC_FMU* fubInstance);

void CNC_FMU_stepFMU(struct CNC_FMU* fubInstance);
void CNC_FMU_resetFMU (struct CNC_FMU* fubInstance);

void CNC_FMU_copyOutputsFromFmu(struct CNC_FMU* fubInstance);
void CNC_FMU_copyInputsToFmu(struct CNC_FMU* fubInstance);
void CNC_FMU_clearFmuOutputs(struct CNC_FMU* fubInstance);

/**********************************************************************/
/* FUB implementation */
void CNC_FMU(struct CNC_FMU* fubInstance)
{
	CNC_FMU_ProcessFmuState(fubInstance);
}

/* Processes the fmu states */
void  CNC_FMU_ProcessFmuState(struct CNC_FMU* fubInstance)
{
	if (FMU_Enable)
	{
		if (!FMU_Enabled)
		{
			CNC_FMU_initFMU(fubInstance);
			FMU_Enabled = fmi2True;
		}

		if(FMU_Error == 0)
		{
			CNC_FMU_stepFMU(fubInstance);
		}
	}else
	{
		if (FMU_Enabled)
		{
			CNC_FMU_resetFMU(fubInstance);
			FMU_Enabled = fmi2False;
		}
	}
	fubInstance->InstRef = &(fubInstance->Internal);
}

/* Initialises the FMU */
void CNC_FMU_initFMU(struct CNC_FMU* fubInstance)
{
	fmi2Status retStatus = fmi2OK;
	FMU_Error = 0;

	CNC_FMU_initFMUCoSimParameters(fubInstance);

	CNC_FMU_initFMUCallbacks(fubInstance);

	FMU_Instance = CNC_FMU_fmi2Instantiate("CNC_FMU",fmi2CoSimulation,"{0f3398f8-206d-0d3a-c8cf-c7c7b11e43f1}",NULL,&FMU_Callbacks,fmi2False,fmi2False);

	if (!FMU_Instance)
	{
		FMU_Error = fmi2True;
	}else
	{
		retStatus = CNC_FMU_fmi2SetupExperiment(FMU_Instance,0 ,0.0, FMU_StartTime, 0, FMU_EndTime);

		if (retStatus > fmi2Warning)
		{
			FMU_Error = fmi2True;
			return;
		}

		retStatus = CNC_FMU_fmi2EnterInitializationMode(FMU_Instance);
		if (retStatus > fmi2Warning)
		{
			FMU_Error = fmi2True;
			return;
		}

		retStatus = CNC_FMU_fmi2ExitInitializationMode(FMU_Instance);
		if (retStatus > fmi2Warning)
		{
			FMU_Error = fmi2True;
			return;
		}

		CNC_FMU_copyOutputsFromFmu(fubInstance);
	}
}

/* Initialize CoSimulation parmeters */
void CNC_FMU_initFMUCoSimParameters(struct CNC_FMU* fubInstance)
{
	FMU_StartTime = 0.00000000000000000e+00;
	FMU_EndTime = 0.0;
	FMU_StepSize = 1.00000000000000000e-04;

	FMU_CurrentTime = 0.0;
}

/* Initialize FMU callbacks */
void  CNC_FMU_initFMUCallbacks(struct CNC_FMU* fubInstance)
{
	FMU_Callbacks.Logger = CNC_FMU_fmuLogger;
	FMU_Callbacks.AllocateMemory = CNC_FMU_AllocateMemory;
	FMU_Callbacks.FreeMemory = CNC_FMU_FreeMemory;
	FMU_Callbacks.StepFinished = NULL;
	FMU_Callbacks.ComponentEnvironment = NULL;
}

/* Execute FMU steps */
void CNC_FMU_stepFMU(struct CNC_FMU* fubInstance)
{

	if (FMU_Error == 0)
	{
		CNC_FMU_copyInputsToFmu(fubInstance);

		fmi2Status retStatus = CNC_FMU_fmi2DoStep(FMU_Instance, FMU_CurrentTime, FMU_StepSize, fmi2True);

		if(retStatus <= fmi2Warning)
		{
			CNC_FMU_copyOutputsFromFmu(fubInstance);

			FMU_CurrentTime += FMU_StepSize;
		}else
		{
			FMU_Error = fmi2True;
		}
	}
}

/* Reset the FMU */
void CNC_FMU_resetFMU (struct CNC_FMU* fubInstance)
{
	fmi2Status retStatus = CNC_FMU_fmi2Reset(FMU_Instance);

	if(retStatus <= fmi2Warning)
	{
		CNC_FMU_clearFmuOutputs(fubInstance);
		FMU_CurrentTime = 0;
	}else
	{
		FMU_Error = fmi2True;
	}
}

/* Log FMU calls */
void CNC_FMU_fmuLogger(void *componentEnvironment, fmi2String instanceName, fmi2Status status, fmi2String category, fmi2String message, ...)
{

}

/* Allocate memory */
void* CNC_FMU_AllocateMemory(UDINT numElements, UDINT elementSize)
{
	void* address;
	UDINT status = 0;

	status = TMP_alloc(numElements * elementSize, &address);

	if (status == 0)
	{
		return address;
	}
	else
	{
		return NULL;
	}
}

/* Free allocated memory */
void CNC_FMU_FreeMemory(void* pMemory)
{
	free(pMemory);
}

/* Clear the output values of the FMU */
void CNC_FMU_clearFmuOutputs(struct CNC_FMU* fubInstance)
{
	/*Clear fmu output PositionX*/
	fubInstance->PositionX = 0.0;
	/*Clear fmu output PositionY*/
	fubInstance->PositionY = 0.0;
	/*Clear fmu output SpeedX*/
	fubInstance->SpeedX = 0.0;
	/*Clear fmu output SpeedY*/
	fubInstance->SpeedY = 0.0;
	/*Clear fmu output TorqueX*/
	fubInstance->TorqueX = 0.0;
	/*Clear fmu output TorqueY*/
	fubInstance->TorqueY = 0.0;

}

/* Copy output values from the FMU */
void CNC_FMU_copyOutputsFromFmu(struct CNC_FMU* fubInstance)
{
	fmi2ValueReference valueReference;
	fmi2Status retStatus = fmi2OK;

	/*Copy fmu output PositionX to PositionX */
	valueReference = 25;
	fmi2Real PositionX;
	retStatus = CNC_FMU_fmi2GetReal(FMU_Instance, &valueReference, 1, &PositionX);

	if(retStatus <= fmi2Warning)
	{
		fubInstance->PositionX = PositionX;
	}else
	{
		FMU_Error = fmi2True;
		return;
	}
	/*Copy fmu output PositionY to PositionY */
	valueReference = 26;
	fmi2Real PositionY;
	retStatus = CNC_FMU_fmi2GetReal(FMU_Instance, &valueReference, 1, &PositionY);

	if(retStatus <= fmi2Warning)
	{
		fubInstance->PositionY = PositionY;
	}else
	{
		FMU_Error = fmi2True;
		return;
	}
	/*Copy fmu output SpeedX to SpeedX */
	valueReference = 2;
	fmi2Real SpeedX;
	retStatus = CNC_FMU_fmi2GetReal(FMU_Instance, &valueReference, 1, &SpeedX);

	if(retStatus <= fmi2Warning)
	{
		fubInstance->SpeedX = SpeedX;
	}else
	{
		FMU_Error = fmi2True;
		return;
	}
	/*Copy fmu output SpeedY to SpeedY */
	valueReference = 4;
	fmi2Real SpeedY;
	retStatus = CNC_FMU_fmi2GetReal(FMU_Instance, &valueReference, 1, &SpeedY);

	if(retStatus <= fmi2Warning)
	{
		fubInstance->SpeedY = SpeedY;
	}else
	{
		FMU_Error = fmi2True;
		return;
	}
	/*Copy fmu output TorqueX to TorqueX */
	valueReference = 27;
	fmi2Real TorqueX;
	retStatus = CNC_FMU_fmi2GetReal(FMU_Instance, &valueReference, 1, &TorqueX);

	if(retStatus <= fmi2Warning)
	{
		fubInstance->TorqueX = TorqueX;
	}else
	{
		FMU_Error = fmi2True;
		return;
	}
	/*Copy fmu output TorqueY to TorqueY */
	valueReference = 28;
	fmi2Real TorqueY;
	retStatus = CNC_FMU_fmi2GetReal(FMU_Instance, &valueReference, 1, &TorqueY);

	if(retStatus <= fmi2Warning)
	{
		fubInstance->TorqueY = TorqueY;
	}else
	{
		FMU_Error = fmi2True;
		return;
	}
}

/* Copy input values to the FMU */
void CNC_FMU_copyInputsToFmu(struct CNC_FMU* fubInstance)
{
	fmi2ValueReference valueReference;
	fmi2Status retStatus = fmi2OK;

	/*Copy fmu input X to X */
	valueReference = 31;
	fmi2Real X;
	X = fubInstance->X;
	retStatus = CNC_FMU_fmi2SetReal(FMU_Instance, &valueReference, 1, &X);
	if(retStatus > fmi2Warning)
	{
		FMU_Error = fmi2True;
		return;
	}
	/*Copy fmu input Y to Y */
	valueReference = 32;
	fmi2Real Y;
	Y = fubInstance->Y;
	retStatus = CNC_FMU_fmi2SetReal(FMU_Instance, &valueReference, 1, &Y);
	if(retStatus > fmi2Warning)
	{
		FMU_Error = fmi2True;
		return;
	}
}
```

### Program Logical/CNC_FMUFmu2/CNC_FMUPrg (ANSIC)

#### Cyclic.c - Cyclic code
```c
#include <bur/plctypes.h>

#ifdef _DEFAULT_INCLUDES
#include <AsDefault.h>
#endif

void _CYCLIC ProgramCyclic(void)
{
	CNC_FMU(&CNC_FMU1);

	CNC_FMUView_0 .InstRef = CNC_FMU1.InstRef;

	CNC_FMUView(&CNC_FMUView_0 );
}
```

#### Init.c - Initialization code
```c
#include <bur/plctypes.h>

#ifdef _DEFAULT_INCLUDES
	#include <AsDefault.h>
#endif

void _INIT ProgramInit(void)
{

}
```

#### Variables.var - Local variables
```iecst
VAR
	CNC_FMU1 : CNC_FMU := (0);
	CNC_FMUView_0 : CNC_FMUView := (0);
END_VAR
```

### Program Logical/CNC_Programs/InitiationandHoming

#### Main.st
```iecst
PROGRAM _INIT
    (*MpCnc2Axis config*)
	MpCnc2Axis_0.MpLink := ADR(gCncXZ);
	MpCnc2Axis_0.Enable := FALSE;
	MpCnc2Axis_0.Parameters := ADR(CncParameters);

	MpCnc2Axis_0.Override := 100.0;
	CncParameters.ProgramName := CncNameCopy;

	(*MpAxisBasic X and Y config*)
	MpAxisBasicX.MpLink:=ADR(gAxisQX);
	MpAxisBasicY.MpLink:=ADR(gAxisQZ);

	MpAxisBasicX.Parameters:=ADR(MpBasicParametersX);
	MpAxisBasicY.Parameters:=ADR(MpBasicParametersY);

	(*--------------------------*)

	MoveMachine := FALSE;

END_PROGRAM

PROGRAM _CYCLIC

	(*Cnc param*)
	CncParameters.Jog.PathLimits.Acceleration	:= gParameter.limit_acc;
	CncParameters.Jog.PathLimits.Deceleration	:= gParameter.limit_dec;
	CncParameters.Jog.PathLimits.Velocity		:= gParameter.limit_vel;
	CncParameters.Jog.Velocity[0]				:= gParameter.set_X_vel;
	CncParameters.Jog.Velocity[1]				:= gParameter.set_Z_vel;

	(*MpAxisBasic param*)
	MpBasicParametersX.Acceleration	:= gParameter.limit_acc;
	MpBasicParametersX.Deceleration	:= gParameter.limit_dec;
	MpBasicParametersX.Velocity		:= gParameter.set_X_vel;

	MpBasicParametersY.Acceleration	:= gParameter.limit_acc;
	MpBasicParametersY.Deceleration	:= gParameter.limit_dec;
	MpBasicParametersY.Velocity		:= gParameter.set_X_vel;

	//Displaying point on manual control screen
	CncPosX:=LREAL_TO_INT(MpCnc2Axis_0.X);
	CncPosY:=LREAL_TO_INT(MpCnc2Axis_0.Y);

	//Start button
	IF ButtonEnable THEN
		MpCnc2Axis_0.Enable := TRUE;
		IF MpCnc2Axis_0.Info.ReadyToPowerOn THEN
			MpCnc2Axis_0.Power := TRUE;
		END_IF;
		IF MpCnc2Axis_0.PowerOn THEN
			MpCnc2Axis_0.Home := TRUE;
		END_IF;
	ELSIF ButtonEnable = FALSE THEN
		gManualContr:=FALSE;
		MpCnc2Axis_0.Enable := FALSE;
		MpCnc2Axis_0.Power := FALSE;

	END_IF;

//Axis enabled after homing and initiation
	IF MpCnc2Axis_0.IsHomed THEN
		MpCnc2Axis_0.Home := FALSE;
		MpAxisBasicX.Enable:=TRUE;
		MpAxisBasicY.Enable:=TRUE;
		MpAxisBasicX.Power:=TRUE;
		MpAxisBasicY.Power:=TRUE;

	END_IF;

//Forcing functions
	MpCnc2Axis_0();
	MpAxisBasicX();
	MpAxisBasicY();

END_PROGRAM

PROGRAM _EXIT

    (*MpCnc2Axis*)

	MpCnc2Axis_0.Power  := FALSE;
	MpCnc2Axis_0.Home   := FALSE;
	MpCnc2Axis_0.Enable := FALSE;
	MpCnc2Axis_0();

	(*MpAxisBasic*)

	MpAxisBasicX.Power  := FALSE;
	MpAxisBasicX.Home   := FALSE;
	MpAxisBasicX.MoveAbsolute := FALSE;
	MpAxisBasicX.MoveAdditive := FALSE;
	MpAxisBasicX.MoveVelocity := FALSE;
	MpAxisBasicX.Stop         := FALSE;
	MpAxisBasicX.ErrorReset   := FALSE;
	MpAxisBasicX();

	MpAxisBasicX.Enable := FALSE;
	MpAxisBasicX();

	MpAxisBasicY.Power  := FALSE;
	MpAxisBasicY.Home   := FALSE;
	MpAxisBasicY.Enable := FALSE;
	MpAxisBasicY.MoveAbsolute := FALSE;
	MpAxisBasicY.MoveAdditive := FALSE;
	MpAxisBasicY.MoveVelocity := FALSE;
	MpAxisBasicY.Stop         := FALSE;
	MpAxisBasicY.ErrorReset   := FALSE;
	MpAxisBasicY();

	MpAxisBasicY.Enable := FALSE;
	MpAxisBasicY();

END_PROGRAM
```

### Program Logical/CNC_Programs/ManualContr

#### Variables.var
```iecst
VAR
	PosY : INT;
	PosX : INT;
	GoDown : BOOL;
	GoRight : BOOL;
	GoLeft : BOOL;
	GoUp : BOOL;
	pointStrX : STRING[80];
	pointStrY : STRING[80];
	strHelp : STRING[80];
	pointString : STRING[120];
	GetThere : BOOL;
END_VAR
```

#### Main.st
```iecst
PROGRAM _INIT

	gStartValueChanging;
	MpCnc2Axis_0;
	CncParameters;
	gActiveTool;

	gMoveAbsoluteX:=TRUE;
	gMoveAbsoluteY:=TRUE;

END_PROGRAM

PROGRAM _CYCLIC

	IF MpCnc2Axis_0.MoveProgram THEN
	  gManualContr:=FALSE;
	END_IF;

	(*When activating manual control*)
	IF EDGEPOS(gManualContr) THEN
	MpBasicParametersX.Position:=MpCnc2Axis_0.X;
	MpBasicParametersY.Position:=MpCnc2Axis_0.Y;
	END_IF

	(*Manual control operating mode switched on with a button in Visu*)
	IF gManualContr THEN

		(*Movement controlled by sliders and text input in visualization*)

		PosX:=LREAL_TO_INT(MpBasicParametersX.Position);
		PosY:=LREAL_TO_INT(MpBasicParametersY.Position);

		IF MpBasicParametersX.Position=INT_TO_LREAL(CncPosX) THEN
			gMoveAbsoluteX:=FALSE;
		END_IF;

		IF MpBasicParametersY.Position=INT_TO_LREAL(CncPosY) THEN
			gMoveAbsoluteY:=FALSE;
		END_IF;

		(*Movement in X (MOVE ABSOLUTE) *)
		IF gMoveAbsoluteX THEN
			MpAxisBasicX.MoveAbsolute:=TRUE;
		END_IF;

		IF MpAxisBasicX.MoveDone=TRUE THEN
			MpAxisBasicX.MoveAbsolute:=FALSE;
			gMoveAbsoluteX:=FALSE;
		END_IF;

		IF EDGENEG(gMoveAbsoluteX) AND CncPosX<>PosX THEN
			gMoveAbsoluteX:=TRUE;
		END_IF;

		(*Movement in Y  (MOVE ABSOLUTE) *)

		IF gMoveAbsoluteY THEN
			MpAxisBasicY.MoveAbsolute:=TRUE;
		END_IF;

		IF MpAxisBasicY.MoveDone=TRUE THEN
			MpAxisBasicY.MoveAbsolute:=FALSE;
			gMoveAbsoluteY:=FALSE;
		END_IF;

		IF EDGENEG(gMoveAbsoluteY) AND CncPosY<>PosY THEN
			gMoveAbsoluteY:=TRUE;
		END_IF;

	ELSIF gManualContr=FALSE THEN
		MpAxisBasicX.MoveAbsolute:=FALSE;
		MpAxisBasicY.MoveAbsolute:=FALSE;
	END_IF;

	(*Movement control with ARROWS in visualization*)

	(*Arrows parameters*)

	MpBasicParametersX.Jog.Velocity:=gParameter.set_X_vel;
	MpBasicParametersY.Jog.Velocity:=gParameter.set_Z_vel;
	MpBasicParametersX.Jog.Acceleration:=gParameter.limit_acc;
	MpBasicParametersY.Jog.Acceleration:=gParameter.limit_acc;
	MpBasicParametersX.Jog.Deceleration:=gParameter.limit_dec;
	MpBasicParametersY.Jog.Deceleration:=gParameter.limit_dec;

	MpBasicParametersX.Jog.LimitPosition.FirstPosition:=0;
	MpBasicParametersX.Jog.LimitPosition.LastPosition:=520;
	MpBasicParametersY.Jog.LimitPosition.FirstPosition:=0;
	MpBasicParametersY.Jog.LimitPosition.LastPosition:=420;

	(*JOG MOVEMENT - NEGATIVE AND POSITIVE*)
	IF MpCnc2Axis_0.MoveActive AND (EDGENEG(MpAxisBasicX.JogNegative) OR EDGENEG(MpAxisBasicY.JogNegative) OR EDGENEG(MpAxisBasicX.JogPositive) OR EDGENEG(MpAxisBasicY.JogPositive)) THEN
	GetThere:=TRUE;
	END_IF;

	IF GetThere THEN
		MpBasicParametersY.Position:=MpCnc2Axis_0.Y;
		MpBasicParametersX.Position:=MpCnc2Axis_0.X;
	END_IF;

	IF MpCnc2Axis_0.MoveActive=FALSE THEN
		GetThere:=FALSE;
	END_IF

	(*Go Up, GoDown, GoLeft and GoRight are variables connected to the arrows in visu*)
	(*UP*)
	IF GoUp=TRUE THEN
		//	MpBasicParametersY.Position:=INT_TO_LREAL(CncPosY);
		MpBasicParametersY.Position:=MpCnc2Axis_0.Y;
		MpAxisBasicY.MoveAbsolute:=FALSE;
		MpAxisBasicY.JogNegative:=TRUE;

	ELSIF GoUp=FALSE THEN
		MpAxisBasicY.JogNegative:=FALSE;
	END_IF;

	(*DOWN*)
	IF GoDown THEN
		MpBasicParametersY.Position:=INT_TO_LREAL(CncPosY);
		MpAxisBasicY.MoveAbsolute:=FALSE;
		MpAxisBasicY.JogPositive:=TRUE;

	ELSIF GoDown=FALSE THEN
		MpAxisBasicY.JogPositive:=FALSE;
	END_IF;

	(*LEFT*)
	IF GoLeft  THEN
		MpBasicParametersX.Position:=INT_TO_LREAL(CncPosX);
		MpAxisBasicX.MoveAbsolute:=FALSE;
		MpAxisBasicX.JogNegative:=TRUE;

	ELSIF GoLeft=FALSE THEN
		MpAxisBasicX.JogNegative:=FALSE;
	END_IF;

		(*RIGHT*)
	IF GoRight THEN
		MpBasicParametersX.Position:=INT_TO_LREAL(CncPosX);
		MpAxisBasicX.MoveAbsolute:=FALSE;
		MpAxisBasicX.JogPositive:=TRUE;

	ELSIF GoRight=FALSE THEN
		MpAxisBasicX.JogPositive:=FALSE;
	END_IF;

	(*Limits for movement in both directions (x,y) *)

	IF MpBasicParametersY.Position>=420 THEN
		MpBasicParametersY.Position:=420;

	ELSIF MpBasicParametersY.Position<=0 THEN
		MpBasicParametersY.Position:=0;
	END_IF;

	IF MpBasicParametersX.Position>=520 THEN
		MpBasicParametersX.Position:=520;

	ELSIF MpBasicParametersX.Position<=0 THEN
		MpBasicParametersX.Position:=0;
	END_IF;

	(* A dot showing the position of the tool*)
	pointString:='<circle cx="';

	pointStrX:=REAL_TO_STRING(CncPosX*1.4);
	pointStrY:=REAL_TO_STRING(CncPosY*1.4);

	strHelp:='" cy="';
	strcat(ADR(pointString),ADR(pointStrX));
	strcat(ADR(pointString),ADR(strHelp));
	strcat(ADR(pointString),ADR(pointStrY));
	strHelp:='" r="5" stroke="black" stroke-width="3" fill="red" />';
	strcat(ADR(pointString),ADR(strHelp));

	MpAxisBasicX();
	MpAxisBasicY();

END_PROGRAM

PROGRAM _EXIT

END_PROGRAM
```

### Program Logical/LibAsIcmp1_ST/Icmp_Ping (IEC) - Example for AsIcmp library

#### Icmp_Ping.st - Cyclic code
```iecst
(********************************************************************
 * COPYRIGHT -- Bernecker + Rainer
 ********************************************************************
 * Program: Icmp_Ping
 * File: Icmp_Ping.st
 * Author: Bernecker + Rainer
 * Created: April 21, 2009
 ********************************************************************
 * Implementation of program Icmp_Ping
 ********************************************************************)

PROGRAM _INIT

	strcpy(ADR(Ping.Host),ADR('216.58.215.110'));

END_PROGRAM

PROGRAM _CYCLIC

	CASE Ping.step OF

		1:	(*Ping station*)
			Ping.IcmpPing_0.enable := 1;  (*Enables the FBK*)
			Ping.IcmpPing_0.pHost := ADR(Ping.Host);  (*IP address or name (SG4 only) of the station (host) that should be pinged*)
			Ping.IcmpPing_0.timeout := 5;  (*Response timeout. Specified in 10ms steps (1 = 10ms, 2 = 20ms, etc.). If 0 is specified, the default timeout (10ms) is used.*)

			Ping.IcmpPing_0;  (*Call FBK*)

			IF Ping.IcmpPing_0.status = 0 THEN  (*FBK finished, go to "wait" step*)
				Ping.step := 2;
			ELSIF Ping.IcmpPing_0.status = ERR_FUB_BUSY THEN  (*FBK still busy, call again*)
				Ping.step := 1;
			ELSE  (*Go to error step*)
				Ping.step := 10;
			END_IF

		2:	(*Wait step*)
			Ping.step := 2;

		10:	(*Here some error handling has to be implemented*)

	END_CASE

END_PROGRAM
```

#### Icmp_Ping.typ - Local data types
```iecst
(********************************************************************
 * COPYRIGHT -- Bernecker + Rainer
 ********************************************************************
 * Program: Icmp_Ping
 * File: Icmp_Ping.typ
 * Author: Bernecker + Rainer
 * Created: April 21, 2009
 ********************************************************************
 * Local data types of program Icmp_Ping
 ********************************************************************)

TYPE
	Ping_typ : 	STRUCT
		step : UINT; (*Step variable*)
		IcmpPing_0 : IcmpPing; (*Function block IcmpPing*)
		Host : STRING[80]; (*Host name*)
	END_STRUCT;
END_TYPE
```

#### Icmp_Ping.var - Local variables
```iecst
(********************************************************************
 * COPYRIGHT -- Bernecker + Rainer
 ********************************************************************
 * Program: Icmp_Ping
 * File: Icmp_Ping.var
 * Author: Bernecker + Rainer
 * Created: April 21, 2009
 ********************************************************************
 * Local variables of program Icmp_Ping
 ********************************************************************)
VAR
	Ping : Ping_typ; (*Variable of Ping_typ*)
END_VAR
```

### Program Logical/LibAsSmtp1_ST/Smtp_Send (IEC) - Example for AsSmtp library

#### Smtp_Send.st - Cyclic code
```iecst
(********************************************************************
 * COPYRIGHT -- Bernecker + Rainer
 ********************************************************************
 * Program: Smtp_Send
 * File: Smtp_Send.st
 * Author: Bernecker + Rainer
 * Created: April 17, 2009
 ********************************************************************
 * Implementation of program Smtp_Send
 ********************************************************************)

PROGRAM _INIT

	strcpy(ADR(Smtp.Parameter.Host),ADR('127.0.0.1'));
	strcpy(ADR(Smtp.Parameter.Sender),ADR('lis.weronika.m@gmail.com'));
	strcpy(ADR(Smtp.Parameter.Receiver),ADR('lis.weronika.m@gmail.com'));	strcpy(ADR(Smtp.Parameter.Subject),ADR('Example mail'));
	strcpy(ADR(Smtp.Parameter.Text),ADR('This text is sent in an email using the AsSmtp library.    Attachment:  '));

END_PROGRAM

PROGRAM _CYCLIC

	CASE Smtp.step OF

		1:	(*Send mail*)
			Smtp.SmtpSend_0.enable := 1;  (*Enables the FBK.*)
			Smtp.SmtpSend_0.pHost := ADR(Smtp.Parameter.Host);  (*IP adress of the SMTP server.*)

			Smtp.SmtpSend_0.pUser := 0;  (*User name, optional. If 0 is specified, authentication does not take place.*)
			Smtp.SmtpSend_0.pPassword := 0;  (*Password,  optional. If 0 is specified, authentication does not take place.*)

			Smtp.SmtpSend_0.pSender := ADR(Smtp.Parameter.Sender);  (*Sender name*)
			Smtp.SmtpSend_0.pReceiver := ADR(Smtp.Parameter.Receiver);  (*Receiver string, can also contain several recipients that are separated by ',' or a space.*)
			Smtp.SmtpSend_0.pSubject := ADR(Smtp.Parameter.Subject);  (*Subject string*)
			Smtp.SmtpSend_0.pText := ADR(Smtp.Parameter.Text);  (*Text string*)

			Smtp.SmtpSend_0.pDomain := 0;  (*Sender domain name, optional, If 0 is specified, "[127.0.0.1]" is entered as the sender domain name.*)

			(*Attachment structure*)
			Smtp.SmtpAttachment.type := smtpATT_TYPE_DATMOD;  (*Type of attachment.*)
			Smtp.SmtpAttachment.pData := ADR('DatObj');  (*Data source of attachment.*)
			Smtp.SmtpAttachment.pName := 0;  (*Name of attachment, optional.*)
			Smtp.SmtpAttachment.length := 0;  (*Length of attachment.*)

			(*Attachment*)
			Smtp.SmtpSend_0.pAttachment := ADR(Smtp.SmtpAttachment);  (*Pointer to attachment structure.*)
			Smtp.SmtpSend_0.attcnt := 1;  (*Number of attachments.*)

			Smtp.SmtpSend_0.timeout := 0;  (*Server response timeout, optional. If 0 is specified, the default timeout of 120s is used.*)
			Smtp.SmtpSend_0.port := 0;  (*Server port number, optional. If 0 is specified, the default port is used (SMTP: 25).*)

			Smtp.SmtpSend_0;  (*Call FBK*)

			IF Smtp.SmtpSend_0.status = 0 THEN  (*FBK finished, go to wait step.*)
				Smtp.step := 2;
			ELSIF Smtp.SmtpSend_0.status = ERR_FUB_BUSY THEN  (*FBK still busy, call again.*)
				Smtp.step := 1;
			ELSE  (*Go to error step.*)
				Smtp.step := 10;
			END_IF

		2:	(*Wait step*)
			Smtp.step := 2;

		10:	(*Here some error handling has to be implemented.*)

	END_CASE

END_PROGRAM
```

#### Smtp_Send.typ - Local data types
```iecst
(********************************************************************
 * COPYRIGHT -- Bernecker + Rainer
 ********************************************************************
 * Program: Smtp_Send
 * File: Smtp_Send.typ
 * Author: Bernecker + Rainer
 * Created: April 17, 2009
 ********************************************************************
 * Local data types of program Smtp_Send
 ********************************************************************)

TYPE
	Smtp_typ : 	STRUCT
		step : UINT; (*Step variable*)
		SmtpSend_0 : SmtpSend; (*Function block SmtpSend*)
		SmtpAttachment : smtpATTACHMENT_typ; (*Attachment variable*)
		Parameter : Parameter_typ; (*Parameter variable*)
	END_STRUCT;
	Parameter_typ : 	STRUCT  (*Parameter structure*)
		Host : STRING[80]; (*Host name*)
		Sender : STRING[80]; (*Name of the sender*)
		Receiver : STRING[80]; (*Name of the receiver*)
		Subject : STRING[80]; (*Subject name*)
		Text : STRING[200]; (*Text in email*)
	END_STRUCT;
END_TYPE
```

#### Smtp_Send.var - Local variables
```iecst
(********************************************************************
 * COPYRIGHT -- Bernecker + Rainer
 ********************************************************************
 * Program: Smtp_Send
 * File: Smtp_Send.var
 * Author: Bernecker + Rainer
 * Created: April 17, 2009
 ********************************************************************
 * Local variables of program Smtp_Send
 ********************************************************************)
VAR
	Smtp : Smtp_typ; (*Variable of Smtp_typ*)
END_VAR
```

### Data object Logical/LibAsSmtp1_ST/DatObj (Simple) - Data object used as email attachment

#### DatObj.dat
```
(********************************************************************
 * COPYRIGHT -- Bernecker + Rainer
 ********************************************************************
 * Data object: DatObj
 * File: DatObj.dat
 * Author: Bernecker + Rainer
 * Created: April 22, 2009
 ********************************************************************
 * Data object file: DatObj.dat
 ********************************************************************)
"Test"
```

### Program Logical/live_drawing/live_draw (IEC)

#### Main.st - Init, cyclic, exit code
```iecst
PROGRAM _INIT

	readX;
	readY;

END_PROGRAM

PROGRAM _CYCLIC

	IF gSvgStringArrayIndex>0 THEN
		gLiveDrawing:=TRUE;
	ELSE
		gLiveDrawing:=FALSE;

	END_IF;

	(*Warning*)

	IF InfoString='Shape outside drawing field!' THEN
		gMsgBox:=TRUE;
	ELSE
		gMsgBox:=FALSE;
	END_IF;

	IF InfoString='Radius can not be equal to 0!' THEN
		gMsgBox2:=TRUE;
	ELSE
		gMsgBox2:=FALSE;
	END_IF;

	IF InfoString='Distance can not be equal to 0!' THEN
		gMsgBox3:=TRUE;
	ELSE
		gMsgBox3:=FALSE;
	END_IF;

	CASE curShape OF
		circle:
			(*-circle drawing-*)
			CASE stage OF
				0:
			InfoString:='Point centre of the circle';
					IF EDGEPOS(cmdDraw) THEN
						cmdDraw:=FALSE;
						shapeString:='<circle cx="';
						prevReadX:=readX;
						prevReadY:=readY;
						strX:=UINT_TO_STRING(readX);
						strY:=UINT_TO_STRING(readY);

						strHelp:='" cy="';
						strcat(ADR(shapeString),ADR(strX));
						strcat(ADR(shapeString),ADR(strHelp));
						strcat(ADR(shapeString),ADR(strY));
						strHelp:='" r="';
						strcat(ADR(shapeString),ADR(strHelp));
						stage:=1;
					END_IF;

				1:
				InfoString:='Point distance from the centre';
					IF EDGEPOS(cmdDraw) THEN
						cmdDraw:=FALSE;
						distX:=ABS(readX-prevReadX);
						distY:=ABS(readY-prevReadY);
						distX:=distX*distX;
						distY:=distY*distY;
						radius:=SQRT(UDINT_TO_REAL(distX+distY));

						IF prevReadX-radius<0 OR prevReadY-radius<0 OR prevReadX+radius>780 OR prevReadY+radius>630 THEN
							stage:=2;
						ELSIF radius=0 THEN
							stage:=3;
						ELSE
							strRadius:=REAL_TO_STRING(radius);
							strcat(ADR(shapeString),ADR(strRadius));
							strHelp:='" stroke="black" fill="none" />';
							strcat(ADR(shapeString),ADR(strHelp));

							svgStringArray[svgStringArrayIndex]:=shapeString;

							svgStringArrayIndex:=svgStringArrayIndex+1;

							stage:=0;
						END_IF;

					END_IF;
				2:
					InfoString:='Shape outside drawing field!';

					IF EDGEPOS(cmdDraw) THEN
						cmdDraw:=FALSE;
						stage:=0;
					END_IF;

				3:
					InfoString:='Radius can not be equal to 0!';
					IF EDGEPOS(cmdDraw) THEN
						cmdDraw:=FALSE;
						stage:=0;
					END_IF;

			END_CASE;

			(*---------------*)
		line:
			(*-line drawing-*)
			CASE stage OF
				0:
					InfoString:='Point first-point of the line';
					IF EDGEPOS(cmdDraw) THEN
						cmdDraw:=FALSE;
						shapeString:='<polyline points="';
						prevReadX:=readX;
						prevReadY:=readY;

						stage:=1;
					END_IF;

				1:
			InfoString:='Point end-point of the line';
					IF EDGEPOS(cmdDraw) THEN
						cmdDraw:=FALSE;
						strPrevX:=UINT_TO_STRING(prevReadX);
						strPrevY:=UINT_TO_STRING(prevReadY);
						strX:=UINT_TO_STRING(readX);
						strY:=UINT_TO_STRING(readY);
						strHelp:=',';
						strcat(ADR(shapeString),ADR(strPrevX));
						strcat(ADR(shapeString),ADR(strHelp));
						strcat(ADR(shapeString),ADR(strPrevY));
						strHelp:=' ';
						strcat(ADR(shapeString),ADR(strHelp));
						strHelp:=',';
						strcat(ADR(shapeString),ADR(strX));
						strcat(ADR(shapeString),ADR(strHelp));
						strcat(ADR(shapeString),ADR(strY));

						strHelp:='" fill="none" stroke="black" />';
						strcat(ADR(shapeString),ADR(strHelp));
						svgStringArray[svgStringArrayIndex]:=shapeString;

						svgStringArrayIndex:=svgStringArrayIndex+1;

						stage:=0;
					END_IF;

			END_CASE;

		(*---------------*)

		rectangle:
			(*-rectangle drawing-*)
			CASE stage OF
				0:
			InfoString:='Point top-left corner of the rectangle';
					IF EDGEPOS(cmdDraw) THEN
						cmdDraw:=FALSE;
						shapeString:='<polyline points="';
						prevReadX:=readX;
						prevReadY:=readY;

						stage:=1;
					END_IF;

				1:
			InfoString:='Point bottom-right corner of the rectangle';
					IF EDGEPOS(cmdDraw) THEN

						cmdDraw:=FALSE;

						IF readX=prevReadX OR readY=prevReadY THEN
							cmdDraw:=FALSE;
							stage:=2;
						ELSE
							strPrevX:=UINT_TO_STRING(prevReadX);
							strPrevY:=UINT_TO_STRING(prevReadY);
							strX:=UINT_TO_STRING(readX);
							strY:=UINT_TO_STRING(readY);
							strHelp:=',';
							strcat(ADR(shapeString),ADR(strPrevX));
							strcat(ADR(shapeString),ADR(strHelp));
							strcat(ADR(shapeString),ADR(strPrevY));
							strHelp:=' ';
							strcat(ADR(shapeString),ADR(strHelp));
							strHelp:=',';
							strcat(ADR(shapeString),ADR(strX));
							strcat(ADR(shapeString),ADR(strHelp));
							strcat(ADR(shapeString),ADR(strPrevY));
							strHelp:=' ';
							strcat(ADR(shapeString),ADR(strHelp));
							strHelp:=',';
							strcat(ADR(shapeString),ADR(strX));
							strcat(ADR(shapeString),ADR(strHelp));
							strcat(ADR(shapeString),ADR(strY));
							strHelp:=' ';
							strcat(ADR(shapeString),ADR(strHelp));
							strHelp:=',';
							strcat(ADR(shapeString),ADR(strPrevX));
							strcat(ADR(shapeString),ADR(strHelp));
							strcat(ADR(shapeString),ADR(strY));

							strHelp:=' ';
							strcat(ADR(shapeString),ADR(strHelp));
							strHelp:=',';
							strcat(ADR(shapeString),ADR(strPrevX));
							strcat(ADR(shapeString),ADR(strHelp));
							strcat(ADR(shapeString),ADR(strPrevY));

							strHelp:='" fill="none" stroke="black" />';
							strcat(ADR(shapeString),ADR(strHelp));
							svgStringArray[svgStringArrayIndex]:=shapeString;

							svgStringArrayIndex:=svgStringArrayIndex+1;

							stage:=0;
						END_IF;

					END_IF;

				2:
					InfoString:='Distance can not be equal to 0!';

					IF EDGEPOS(cmdDraw) THEN
						cmdDraw:=FALSE;
						stage:=0;
					END_IF;

			END_CASE;

		(*---------------*)

		star:
			(*-star drawing-*)
			CASE stage OF
				0:
				InfoString:='Point centre of the star';
					IF EDGEPOS(cmdDraw) THEN
						cmdDraw:=FALSE;
						shapeString:='<polyline points="';
						prevReadX:=readX;
						prevReadY:=readY;

						stage:=1;
					END_IF;

				1:
				InfoString:='Point distance from the centre';
					IF EDGEPOS(cmdDraw) THEN
						cmdDraw:=FALSE;
						distX:=ABS(readX-prevReadX);
						distY:=ABS(readY-prevReadY);
						distX:=distX*distX;
						distY:=distY*distY;
						radius:=SQRT(UDINT_TO_REAL(distX+distY));
						IF prevReadX-radius<0 OR prevReadY-radius<0 OR prevReadX+radius>780 OR prevReadY+radius>630 THEN
							stage:=2;
						ELSIF radius=0 THEN
							stage:=3;
						ELSE
						smallRadius:=radius/3;
						angle:=-18; // degrees
						FOR i:=1 TO 5 DO

							x:=radius*COS(angle/180*PI);
							y:=radius*SIN(angle/180*PI);
							strX:=REAL_TO_STRING(x+prevReadX);
							strY:=REAL_TO_STRING(y+prevReadY);
							strHelp:=',';
							strcat(ADR(shapeString),ADR(strX));
							strcat(ADR(shapeString),ADR(strHelp));
							strcat(ADR(shapeString),ADR(strY));
							strHelp:=' ';
							strcat(ADR(shapeString),ADR(strHelp));

							x:=smallRadius*COS((angle+36)/180*PI);
							y:=smallRadius*SIN((angle+36)/180*PI);

							strX:=REAL_TO_STRING(x+prevReadX);
							strY:=REAL_TO_STRING(y+prevReadY);
							strHelp:=',';
							strcat(ADR(shapeString),ADR(strX));
							strcat(ADR(shapeString),ADR(strHelp));
							strcat(ADR(shapeString),ADR(strY));
							strHelp:=' ';
							strcat(ADR(shapeString),ADR(strHelp));
							angle:=angle+72;

						END_FOR;

						x:=radius*COS(angle/180*PI);
						y:=radius*SIN(angle/180*PI);
						strX:=REAL_TO_STRING(x+prevReadX);
						strY:=REAL_TO_STRING(y+prevReadY);
						strHelp:=',';
						strcat(ADR(shapeString),ADR(strX));
						strcat(ADR(shapeString),ADR(strHelp));
						strcat(ADR(shapeString),ADR(strY));

						strHelp:='" fill="none" stroke="black" />';
						strcat(ADR(shapeString),ADR(strHelp));
						svgStringArray[svgStringArrayIndex]:=shapeString;

						svgStringArrayIndex:=svgStringArrayIndex+1;

							stage:=0;
							END_IF
					END_IF;
				2:
					InfoString:='Shape outside drawing field!';
					IF EDGEPOS(cmdDraw) THEN
						cmdDraw:=FALSE;
						stage:=0;
					END_IF

				3:
					InfoString:='Distance can not be equal to 0!';
					IF EDGEPOS(cmdDraw) THEN
						cmdDraw:=FALSE;
						stage:=0;
					END_IF;

			END_CASE;

		(*---------------*)

		arc:
			(*-arc drawing-*)
			CASE stage OF
				0:
					InfoString:='Point first-point of the arc';
					IF EDGEPOS(cmdDraw) THEN
						cmdDraw:=FALSE;
						shapeString:='<path d="M ';
						prevPrevReadX:=readX;
						prevPrevReadY:=readY;

						stage:=1;
					END_IF;

				1:
					InfoString:='Point endt-point of the arc';
					IF EDGEPOS(cmdDraw) THEN
						cmdDraw:=FALSE;
						prevReadX:=readX;
						prevReadY:=readY;
						stage:=2;
					END_IF;
				2:
					InfoString:='Point radius distance of the arc';
					IF EDGEPOS(cmdDraw) THEN
						cmdDraw:=FALSE;

						ab:=SQRT(ABS(prevReadX-prevPrevReadX)*ABS(prevReadX-prevPrevReadX)+ABS(prevReadY-prevPrevReadY)*ABS(prevReadY-prevPrevReadY));
						bc:=SQRT(ABS(readX-prevReadX)*ABS(readX-prevReadX)+ABS(readY-prevReadY)*ABS(readY-prevReadY));
						maks:=ab/2;
						radius:=bc;
						IF prevReadX-radius<0 OR prevReadY-radius<0 OR prevReadX+radius>780 OR prevReadY+radius>630 THEN
							stage:=3;
						ELSE

							IF radius> maks THEN
								radius:=maks;
							ELSE
								radius:=(maks*15)-(radius/maks)*(maks*15);

							END_IF

							strHelp:=' ';
							strX:=UINT_TO_STRING(prevPrevReadX);
							strcat(ADR(shapeString),ADR(strX));
							strcat(ADR(shapeString),ADR(strHelp));
							strY:=UINT_TO_STRING(prevPrevReadY);
							strcat(ADR(shapeString),ADR(strY));
							strHelp:=' A ';
							strcat(ADR(shapeString),ADR(strHelp));
							strRadius:=REAL_TO_STRING(radius);
							strcat(ADR(shapeString),ADR(strRadius));
							strHelp:=' ';
							strcat(ADR(shapeString),ADR(strHelp));
							strcat(ADR(shapeString),ADR(strRadius));
							strHelp:=' 0 0 0 ';
							strcat(ADR(shapeString),ADR(strHelp));
							strX:=UINT_TO_STRING(prevReadX);
							strcat(ADR(shapeString),ADR(strX));
							strHelp:=' ';
							strcat(ADR(shapeString),ADR(strHelp));
							strY:=UINT_TO_STRING(prevReadY);
							strcat(ADR(shapeString),ADR(strY));
							strHelp:='" fill="none" stroke="black" />';
							strcat(ADR(shapeString),ADR(strHelp));

							svgStringArray[svgStringArrayIndex]:=shapeString;

							svgStringArrayIndex:=svgStringArrayIndex+1;

							stage:=0;
						END_IF;
						END_IF
				3:
					InfoString:='Shape outside drawing field!';
					IF EDGEPOS(cmdDraw) THEN
						cmdDraw:=FALSE;
						stage:=0;
					END_IF

			END_CASE;

		(*---------------*)

	END_CASE
(*----clearing paper-----*)
	IF EDGEPOS(cmdClear) THEN
		cmdClear:=FALSE;
		FOR i:=0 TO svgStringArrayIndex DO
			svgStringArray[i]:='';
		END_FOR;
		svgStringArrayIndex:=0;
	END_IF;
(*------Undo--------*)
	IF EDGEPOS(cmdBack) THEN
		cmdBack:=FALSE;
		IF svgStringArrayIndex>0 THEN
			svgStringArrayIndex:=svgStringArrayIndex-1;
		END_IF
			svgStringArray[svgStringArrayIndex]:='';

	END_IF;
(*------Pass to global---------*)
	gSvgStringArray:=svgStringArray;
	gSvgStringArrayIndex:=svgStringArrayIndex;

	(*------- Mirroring --------*)

//	IF EDGEPOS(cmdMirror) THEN
//
//	svgString:=gSvgStringArray[0];
//	labelString:=LEFT(svgString,4);
//	Xstr:='';
//	Ystr:='';
//
//	IF labelString='<pol' THEN
//		j:=19;
//		pos:=j;
//		flag1:=TRUE;
//
//		WHILE flag1 DO
//			buff:=MID(svgString,1,j);
//
//
//			IF buff=',' THEN
//				xory:=TRUE;
//
//
//			ELSIF buff=' ' OR buff='"' THEN
//				xory:=FALSE;
//
//				Xreal:=STRING_TO_REAL(Xstr);
//
//				Yreal:=STRING_TO_REAL(Ystr);
//				Xreal:=Xreal+50;
//				Yreal:=Yreal+50;
//
//
//
//			Xstr2:=REAL_TO_STRING(Xreal);
//				Ystr2:=REAL_TO_STRING(Yreal);
//
//				svgString:=REPLACE(svgString,Xstr2,LEN(Xstr),pos);
//				svgString:=REPLACE(svgString,Ystr2,LEN(Ystr),pos+1+LEN(Xstr));
//
//
//				Xstr:='';
//				Ystr:='';
//				pos:=j+1;
//
//				IF buff='"' THEN
//					flag1:=FALSE;
//				END_IF
//
//
//			ELSE
//				IF xory THEN
//					strcat(ADR(Ystr),ADR(buff));
//				ELSE
//
//					strcat(ADR(Xstr),ADR(buff));
//				END_IF
//			END_IF
//			j:=j+1;
//		END_WHILE;
//
//	END_IF
//	END_IF

END_PROGRAM

PROGRAM _EXIT
	(* Insert code here *)

END_PROGRAM
```

#### Variables.var - Local variables
```iecst
VAR
	ab : REAL;
	angle : REAL;
	bc : REAL;
	buff : STRING[80];
	cmdBack : BOOL;
	cmdClear : BOOL;
	cmdDraw : BOOL;
	cmdMirror : BOOL;
	curShape : shape_enum;
	distX : UDINT;
	distY : UDINT;
	flag1 : BOOL;
	i : UINT;
	InfoString : STRING[300];
	j : INT;
	labelString : STRING[80];
	maks : REAL;
END_VAR
VAR CONSTANT
	PI : REAL := 3.141592;
END_VAR
VAR
	pos : INT;
	prevPrevReadX : UINT;
	prevPrevReadY : UINT;
	prevReadX : UINT;
	prevReadY : UINT;
	radius : REAL;
	readX : UINT;
	readY : UINT;
	shapeString : STRING[500];
	smallRadius : REAL;
	stage : INT;
	strHelp : STRING[80];
	strPrevX : STRING[80];
	strPrevY : STRING[80];
	strRadius : STRING[80];
	strX : STRING[80];
	strY : STRING[80];
	svgString : STRING[160];
	svgStringArray : ARRAY[0..999] OF STRING[500];
	svgStringArrayIndex : UINT;
	x : REAL;
	xory : BOOL;
	Xreal : REAL;
	Xstr : STRING[80];
	Xstr2 : STRING[80];
	y : REAL;
	Yreal : REAL;
	Ystr : STRING[80];
	Ystr2 : STRING[80];
END_VAR
```

### Program Logical/live_drawing/svg_to_gcode (IEC)

#### Main.st
```iecst
PROGRAM _INIT
	(* Insert code here *)
	strDevice:= 'CNC_PrgDir';
	strFile:= 'obrazek.cnc';
	bOK := FALSE;
	byStep := 1;
	byErrorLevel := 0;

memset(ADR(cncString), 0, SIZEOF(cncString));
END_PROGRAM

PROGRAM _CYCLIC
	(* Insert code here *)

	IF cmdConvert THEN

		cmdConvert:=FALSE;
		IF gSvgStringArray[0]<>'' THEN

		memset(ADR(cncString), 0, SIZEOF(cncString));
		strHelp:='%001$n';
		strcat(ADR(cncString),ADR(strHelp));
		FOR i:=0 TO (gSvgStringArrayIndex-1) DO

			svgString:=gSvgStringArray[i];
			labelString:=LEFT(svgString,4);
			Xstr:='';
			Ystr:='';
			Rstr:='';
			IF labelString='<pol' THEN
				j:=19;
				flag1:=TRUE;
				firstMove:=TRUE;
				WHILE flag1 DO
					buff:=MID(svgString,1,j);

					IF buff=',' THEN
						xory:=TRUE;

					ELSIF buff=' ' OR buff='"' THEN
						xory:=FALSE;

						Xscale:=STRING_TO_REAL(Xstr)/1.5;
						Xstr:=REAL_TO_STRING(Xscale);
						Yscale:=STRING_TO_REAL(Ystr)/1.5;
						Ystr:=REAL_TO_STRING(Yscale);

						IF firstMove THEN
							IF prevXstr<>Xstr OR prevYstr<>Ystr THEN
								strHelp:='M50$n';    //podniesienie

								strcat(ADR(cncString),ADR(strHelp));

								strHelp:='G01 X';
								strcat(ADR(cncString),ADR(strHelp));
								strcat(ADR(cncString),ADR(Xstr));
								strHelp:=' Z';
								strcat(ADR(cncString),ADR(strHelp));
								strcat(ADR(cncString),ADR(Ystr));
								strHelp:=' F';
								strcat(ADR(cncString),ADR(strHelp));
								strcat(ADR(cncString),ADR(Fstr));
								strHelp:='$n';
								strcat(ADR(cncString),ADR(strHelp));

								strHelp:='M60$n';    //opuszczenie

								strcat(ADR(cncString),ADR(strHelp));
							END_IF
							firstMove:=FALSE;
						ELSE
							strHelp:='G01 X';
							strcat(ADR(cncString),ADR(strHelp));
							strcat(ADR(cncString),ADR(Xstr));
							strHelp:=' Z';
							strcat(ADR(cncString),ADR(strHelp));
							strcat(ADR(cncString),ADR(Ystr));
							strHelp:=' F';
							strcat(ADR(cncString),ADR(strHelp));
							strcat(ADR(cncString),ADR(Fstr));
							strHelp:='$n';
							strcat(ADR(cncString),ADR(strHelp));
						END_IF

						prevXstr:=Xstr;
						prevYstr:=Ystr;

						Xstr:='';
						Ystr:='';

						IF buff='"' THEN
							flag1:=FALSE;
						END_IF

					ELSE
						IF xory THEN
							strcat(ADR(Ystr),ADR(buff));
						ELSE

							strcat(ADR(Xstr),ADR(buff));
						END_IF
					END_IF
					j:=j+1;
				END_WHILE;

			ELSIF labelString='<cir' THEN
				j:=12;
				flag1:=TRUE;
				k:=0;
				WHILE flag1 DO
					buff:=MID(svgString,1,j);

					IF buff='"' THEN

						k:=k+1;
					ELSE

					CASE k OF
						1:

							strcat(ADR(Xstr),ADR(buff));
						3:
							strcat(ADR(Ystr),ADR(buff));
						5:
							strcat(ADR(Rstr),ADR(buff));
							6:	flag1:=FALSE;
								strHelp:='M50$n';    //podniesienie
								Xscale:=STRING_TO_REAL(Xstr)/1.5;
								Xstr:=REAL_TO_STRING(Xscale);
								Yscale:=STRING_TO_REAL(Ystr)/1.5;
								Ystr:=REAL_TO_STRING(Yscale);
								Rscale:=STRING_TO_REAL(Rstr)/1.5;
								Rstr:=REAL_TO_STRING(Rscale);

								Xstr:=REAL_TO_STRING(STRING_TO_REAL(Xstr)-STRING_TO_REAL(Rstr));

								strcat(ADR(cncString),ADR(strHelp));
								strHelp:='G01 X';
								strcat(ADR(cncString),ADR(strHelp));
								strcat(ADR(cncString),ADR(Xstr));
								strHelp:=' Z';
								strcat(ADR(cncString),ADR(strHelp));
								strcat(ADR(cncString),ADR(Ystr));
								strHelp:=' F';
								strcat(ADR(cncString),ADR(strHelp));
								strcat(ADR(cncString),ADR(Fstr));
								strHelp:='$n';
								strcat(ADR(cncString),ADR(strHelp));
								strHelp:='M60$n';    //opuszczenie
								strcat(ADR(cncString),ADR(strHelp));
								strHelp:='G02 I';
								strcat(ADR(cncString),ADR(strHelp));
								strcat(ADR(cncString),ADR(Rstr));
								strHelp:=' H360$n';
								strcat(ADR(cncString),ADR(strHelp));
								Xstr:='';
								Ystr:='';
								Rstr:='';

					END_CASE;
					END_IF

					j:=j+1;
				END_WHILE;

			ELSIF labelString='<pat' THEN
				j:=11;
				flag1:=TRUE;
				k:=0;
				WHILE flag1 DO
					buff:=MID(svgString,1,j);

					IF buff=' ' THEN

						k:=k+1;

					ELSIF buff='"' THEN
						flag1:=FALSE;
						Xscale:=STRING_TO_REAL(Xstr)/1.5;
						Xstr:=REAL_TO_STRING(Xscale);
						Yscale:=STRING_TO_REAL(Ystr)/1.5;
						Ystr:=REAL_TO_STRING(Yscale);

						X2scale:=STRING_TO_REAL(Xstr2)/1.5;
						Xstr2:=REAL_TO_STRING(X2scale);
						Y2scale:=STRING_TO_REAL(Ystr2)/1.5;
						Ystr2:=REAL_TO_STRING(Y2scale);

						Rscale:=STRING_TO_REAL(Rstr)/1.5;
						Rstr:=REAL_TO_STRING(Rscale);
						IF prevXstr<>Xstr OR prevYstr<>Ystr THEN
							strHelp:='M50$n';    //podniesienie

							strcat(ADR(cncString),ADR(strHelp));
							strHelp:='G01 X';
							strcat(ADR(cncString),ADR(strHelp));
							strcat(ADR(cncString),ADR(Xstr));
							strHelp:=' Z';
							strcat(ADR(cncString),ADR(strHelp));
							strcat(ADR(cncString),ADR(Ystr));
							strHelp:=' F';
							strcat(ADR(cncString),ADR(strHelp));
							strcat(ADR(cncString),ADR(Fstr));
							strHelp:='$n';
							strcat(ADR(cncString),ADR(strHelp));
							strHelp:='M60$n';    //opuszczenie
							strcat(ADR(cncString),ADR(strHelp));

						END_IF

						strHelp:='G03 X';
						strcat(ADR(cncString),ADR(strHelp));
						strcat(ADR(cncString),ADR(Xstr2));
						strHelp:=' Z';
						strcat(ADR(cncString),ADR(strHelp));
						strcat(ADR(cncString),ADR(Ystr2));
						strHelp:=' R=';
						strcat(ADR(cncString),ADR(strHelp));
						strcat(ADR(cncString),ADR(Rstr));
						strHelp:='$n';
						strcat(ADR(cncString),ADR(strHelp));
						prevXstr:=Xstr2;
						prevYstr:=Ystr2;

						Xstr:='';
						Ystr:='';
						Rstr:='';
						Xstr2:='';
						Ystr2:='';

					ELSE

						CASE k OF
							1:

								strcat(ADR(Xstr),ADR(buff));
							2:
								strcat(ADR(Ystr),ADR(buff));
							4:
								strcat(ADR(Rstr),ADR(buff));
							9:	strcat(ADR(Xstr2),ADR(buff));

							10:	strcat(ADR(Ystr2),ADR(buff));

						END_CASE;
					END_IF

					j:=j+1;
				END_WHILE;
			END_IF;

		END_FOR;
		strHelp:='M30';
		strcat(ADR(cncString),ADR(strHelp));
		cmdFile:=TRUE;
		END_IF;
	END_IF

						IF cmdFile THEN

						CASE byStep OF
							0: (**** Error step ****)                bOK := FALSE;
							1: (**** Try to open existing file ****)
								(* Initialize file open structrue *)
								FOpen.enable    := 1;
								FOpen.pDevice   := ADR(strDevice);
								FOpen.pFile     := ADR(strFile);
								FOpen.mode      := FILE_RW;  (* Read and write access *)
								(* Call FBK *)                FOpen();
								(* Get FBK output information *)
								dwIdent := FOpen.ident;                wStatus := FOpen.status;
								(* Verify status (20708 -> File doesn't exist) *)
				IF (wStatus = 20708) THEN
					byStep := 2;
					fileFlag:=FALSE;
								ELSE                        IF (wStatus = 0) THEN
						byStep := 5;
						fileFlag:=TRUE;
					ELSE
										IF (wStatus <> 65535) THEN
											byErrorLevel := 1;
											byStep := 0;
											IF (wStatus = 20799) THEN
												wError := FileIoGetSysError();
							END_IF
					END_IF                        END_IF
				END_IF
			2: (**** Create file ****)
				(* Initialize file create structure *)
				FCreate.enable  := 1;
				FCreate.pDevice := ADR(strDevice);
				FCreate.pFile   := ADR(strFile);                (* Call FBK *)
				FCreate();                (* Get FBK output information *)
				dwIdent := FCreate.ident;
				wStatus := FCreate.status;                (* Verify status *)
				IF (wStatus = 0) THEN                        byStep := 3;
				ELSE                        IF (wStatus <> 65535) THEN
						byErrorLevel := 2;
						byStep := 0;
						IF (wStatus = 20799) THEN
							wError := FileIoGetSysError();
					END_IF                        END_IF
				END_IF
			3: (**** Write data to file ****)
				(* Initialize file write structure *)
				FWrite.enable   := 1;               FWrite.ident    := dwIdent;
				FWrite.offset   := 0;
				FWrite.pSrc     := ADR(cncString);
				FWrite.len      := LEN(cncString);
				(* Call FBK *)                FWrite();

				(* Get status *)                wStatus := FWrite.status;
				(* Verify status *)                IF (wStatus = 0) THEN
				byStep := 5;                ELSE
					IF (wStatus <> 65535) THEN
						byErrorLevel := 3;
						byStep := 0;
						IF (wStatus = 20799) THEN
							wError := FileIoGetSysError();
					END_IF                        END_IF
				END_IF
				//		4: (**** Read data from file ****)
				//			(* Initialize file read structure *)
				//			FRead.enable    := 1;                FRead.ident     := dwIdent;
				//			FRead.offset    := 0;
				//			FRead.pDest     := ADR(byReadData[0]);
				//			FRead.len       := SIZEOF(byReadData);
				//			(* Call FBK *)                FRead();
				//			(* Get status *)                wStatus := FRead.status;
				//			(* Verify status *)                IF (wStatus = 0) THEN
				//			byStep := 5;                ELSE
				//				IF (wStatus <> 65535) THEN
				//					byErrorLevel := 4;
				//					byStep := 0;
				//					IF (wStatus = 20799) THEN
				//						wError := FileIoGetSysError();
				//				END_IF                        END_IF
				//			END_IF
			5: (**** Close file ****)
				(* Initialize file close structure *)
				FClose.enable   := 1;                FClose.ident    := dwIdent;
				(* Call FBK *)                FClose();
				(* Get status *)                wStatus := FClose.status;
				(* Verify status *)
				IF (wStatus = 0) THEN

					IF fileFlag THEN

					ELSE

						cmdFile:=FALSE;
						memset(ADR(cncString), 0, SIZEOF(cncString));
					END_IF
					byStep := 1;
					fileIndex:=fileIndex+1;
					strNum:=INT_TO_STRING(fileIndex);
					strFile:='obrazek.cnc';
					strFile := INSERT(strFile, strNum, 7);

				ELSE
					IF (wStatus <> 65535) THEN
						byErrorLevel := 5;
						byStep := 0;

						IF (wStatus = 20799) THEN
							wError := FileIoGetSysError();
					END_IF                        END_IF
				END_IF
			//		6: (**** Delete file ****)
			//			(* Initialize file delete structure *)
			//			FDelete.enable  := 1;
			//			FDelete.pDevice := ADR(strDevice);
			//			FDelete.pName   := ADR(strFile);                (* Call FBK *)
			//			FDelete();                (* Get status *)
			//			wStatus := FDelete.status;                (* Verify status *)
			//			IF (wStatus = 0) THEN                        bOK     := TRUE;
			//			byStep := 7;                ELSE
			//				IF (wStatus <> 65535) THEN
			//					byErrorLevel := 6;
			//					byStep := 0;
			//					IF (wStatus = 20799) THEN
			//						wError := FileIoGetSysError();
			//					END_IF
			//				END_IF
			//			END_IF
		END_CASE

	END_IF

END_PROGRAM

PROGRAM _EXIT
	(* Insert code here *)

END_PROGRAM
```

### Program Logical/Recipe

#### Variables.var
```iecst
VAR
	i : UINT;
	j : UINT;
	k : INT;
	MpRecipeRegPar_0 : MpRecipeRegPar;
	MpRecipeUI_0 : MpRecipeUI;
	MpRecipeXml_0 : MpRecipeXml;
	nextAddr : UDINT;
	TempLine : ARRAY[0..4] OF STRING[80];
	UIConnect : MpRecipeUIConnectType := (Recipe:=(SortOrder:=mpRECIPE_UI_SORT_DATE_ASCENDING));
	UISetup : MpRecipeUISetupType := (RecipeListSize:=5);
	DataProvider0 : ARRAY[0..4] OF STRING[100];
	input : BOOL;
	TP_01 : TP;
	CreatingRecipe : BOOL;
END_VAR
```
